(* 1 - During reseting, 0 - Reset completed
	Description:
		Reset the batetery replacement timer request.
		Indirectly resets the battery error. *) 
METHOD MR_BatteryReset : BOOL
IF NOT BatteryResetCompleted THEN
	bBusy 	:= TRUE;
	MR_BatteryReset := TRUE;
	BatteryReset :=	TRUE;
	fbMachineLogger.MR_AddLogs(CONCAT(sName,' : battery reset requested'));
	
ELSE 
	MR_BatteryReset := FALSE;
	BatteryReset :=	FALSE;
	bBusy 	:= FALSE;
	fbMachineLogger.MR_AddLogs(CONCAT(sName,' : battery reset done'));
	
END_IF
END_METHOD

(* 1 - Cycle paused, 0 - Cycle not paused
	Description:
		This method stop the program without reseting.
		IE. stops movement implicily 
		To restore the movement use MR_RestoreCycle or MR_GoHome *)
METHOD MR_CyclePause : BOOL
IF eCR800State = CR800_DOING_ACTION THEN
	bBusy 	:= TRUE;
	bCyclePause := TRUE;
	MR_CyclePause := FALSE;
	eCR800State := E_CR800State.CR800_CYCLE_PAUSING;
	fbMachineLogger.MR_AddLogs(CONCAT(sName,' : cycle pausing requested'));
	
ELSIF eCR800State = E_CR800State.CR800_CYCLE_PAUSING_DONE THEN
	bCyclePause	:= FALSE;
	MR_CyclePause := TRUE;
	bBusy 	:= FALSE;
	fbMachineLogger.MR_AddLogs(CONCAT(sName,' : cycle pausing done'));
	
END_IF
END_METHOD

(* 1 - During stopping, 0 - Cycle stop completed
	Description:
		This method stop the program, when the "End" command is met in the robots program.
		Caution: It stops the program AND reset it. To restore it you need to use MR_RestoreAuto. *) 

METHOD MR_CycleStop : BOOL
IF eCR800State = CR800_DOING_ACTION OR eCR800State = CR800_IDLE_CYCLE_PAUSED OR eCR800State = CR800_IDLE_AUTO_PAUSED THEN
	bBusy 	:= TRUE;
	bCycleStop 	:= TRUE;
	MR_CycleStop := FALSE;
	eCR800State := CR800_CYCLE_STOPPING;
	fbMachineLogger.MR_AddLogs(CONCAT(sName,' : cycle stopping requested'));
	
ELSIF eCR800State = CR800_CYCLE_STOPING_DONE THEN
	bDoAction := FALSE;
	bCycleStop := FALSE;
	MR_CycleStop := TRUE;
	bBusy 	:= FALSE;
	fbMachineLogger.MR_AddLogs(CONCAT(sName,' : cycle stopping done'));
	
END_IF
END_METHOD

(* 0 - Action not completed, 1 - Action completed
Description:
This method send request to do an action.
Robot will perform an action number that is called in input.
If the action is single and has and end use:
	IF MR_DoAction( iActionNumber := iExampleNumber) THEN
		bDO_A_FLIP := true ;
	END_IF
If the action is endless then just call it, and then use MR_CycleStop.
	MR_DoAction( iActionNumber := iExampleNumber) *)
METHOD MR_DoAction : BOOL
VAR_INPUT
	iActionNumber : UINT ;
END_VAR
IF eCR800State = CR800_IDLE_AUTO THEN
	IF iActionNumber <= 12 THEN 
		bError := TRUE ;
		eErrorID := CR800_ERROR_CANT_DO_SYSTEM_ACTION_IN_THIS_REQUEST ;
	ELSE
		bBusy 	:= TRUE;
		bDoAction := TRUE;
		bStopped := FALSE;
		MR_DoAction := FALSE;
		iActionNumber := iActionNumber;
		eCR800State := CR800_DOING_ACTION;
		fbMachineLogger.MR_AddLogs(FUN_MergeStrings5(sName,' : doing action number: ',UINT_TO_STRING(iActionNumber), '',' requested'));
	
	END_IF
	
ELSIF eCR800State = CR800_DOING_ACTION_DONE THEN
	bIsHomed := FALSE;
	bAutoModeStarted := FALSE;
	MR_DoAction := TRUE;
	bBusy := FALSE; 
	fbMachineLogger.MR_AddLogs(FUN_MergeStrings5(sName,' : doing action number: ',UINT_TO_STRING(iActionNumber),'',' done'));
	
ELSIF eCR800State <> CR800_DOING_ACTION AND eCR800State = E_CR800State.CR800_IDLE_CYCLE_PAUSED 
	AND eCR800State <> E_CR800State.CR800_CYCLE_PAUSING AND eCR800State <> E_CR800State.CR800_CYCLE_PAUSING
	AND eCR800State <> CR800_CYCLE_RESTORING AND eCR800State <> CR800_CYCLE_RESTORING_DONE THEN
	bError := TRUE ;
	eErrorID := CR800_ERROR_CANT_DO_ACTION_WITHOUT_BEEING_AUTO ;
	fbMachineLogger.MR_AddLogs(CONCAT(sName,' : ERROR_CANT_DO_ACTION_WITHOUT_BEEING_AUTO'));
	
END_IF
END_METHOD

METHOD MR_FirstCycle : BOOL
VAR_INPUT
	sName 				: STRING;
	iOverride			: USINT;
END_VAR
THIS^.sName := sName;
THIS^.iOverride := iOverride;
END_METHOD

(* 0 - FB is NOT in auto mode, 1 - FB is in auto mode
	Description:
		This method reqest FB to go into the auto mode. In automode FB can perform actions (MR_DoAction) *)
METHOD MR_GoAuto : BOOL
IF NOT bIsHomed THEN 
	bError := TRUE ;
	eErrorID := CR800_ERROR_CANT_GO_AUTO_WITHOUT_BEEING_HOMED ;
	fbMachineLogger.MR_AddLogs(CONCAT(sName,' : ERROR_CANT_GO_AUTO_WITHOUT_BEEING_HOMED'));
	
ELSIF eCR800State = CR800_IDLE_HOMED OR eCR800State = CR800_CYCLE_PAUSING_IDLE THEN
	bBusy 	:= TRUE;
	bGoAuto := TRUE;
	MR_GoAuto := FALSE;
	iActionNumber := stRobot.iActionNumber;
	eCR800State := CR800_GOING_AUTO;
	fbMachineLogger.MR_AddLogs(CONCAT(sName,' : going auto requested'));
	
ELSIF eCR800State = CR800_GOING_AUTO_DONE THEN
	bStopped := FALSE;
	bGoAuto := FALSE;
	MR_GoAuto := TRUE;
	bAutoModeStarted := TRUE;
	bBusy 	:= FALSE;
	fbMachineLogger.MR_AddLogs(CONCAT(sName,' : going auto done'));
	
END_IF
END_METHOD

(* 1 - Homing finished, 0 - Homing not finished.
	Description:
	This method request the robot to go home *)
METHOD MR_GoHome : BOOL
IF eCR800State = CR800_IDLE_NOT_HOMED OR eCR800State = CR800_IDLE_AUTO OR eCR800State = CR800_IDLE_AUTO_PAUSED THEN
	bBusy 	:= TRUE;	
	bGoHome := TRUE;
	MR_GoHome := FALSE;
	eCR800State := CR800_GOING_HOME;
	fbMachineLogger.MR_AddLogs(CONCAT(sName,' : going home requested'));
	
ELSIF eCR800State = CR800_GOING_HOME_DONE THEN
	bIsHomed := TRUE;
	bGoHome := FALSE;
	MR_GoHome := TRUE;
	bBusy 	:= FALSE;
	fbMachineLogger.MR_AddLogs(CONCAT(sName,' : going home done'));
	
END_IF
END_METHOD

(* 1 - Initializing finished, 0 - Initializing not finished.
	Description:
		This method initialize the robot:
			1. Checks for ethercat connection
			2. Checks for power of the CR800
			3. Checks for emergency stop
			4. Checks is CR800 is in auto mode
			5. Enable rights
			6. Turn on servos
			7. Resets the program
			8. Starts the program
			9. Sets initial parameters in the robot (when initializing after error this step is ommited) *)
METHOD MR_Init : BOOL
IF eCR800State = CR800_UNINITIALIZED AND NOT bAbort AND NOT bReset THEN
	bBusy 	:= TRUE;
	bInit := TRUE;
	MR_Init := FALSE;
	eCR800State := CR800_INITIALIZING;
	fbMachineLogger.MR_AddLogs(CONCAT(sName,' : initialization requested'));
	
ELSIF eCR800State = CR800_READY_INITIALIZED THEN
	bUninitialized := FALSE;
	bActive := TRUE;
	bInit := FALSE;
	MR_Init := TRUE;
	bBusy 	:= FALSE;
	fbMachineLogger.MR_AddLogs(CONCAT(sName,' : initialization done'));
	
END_IF
END_METHOD

(* 1 - Reset finished, 0 - Reset not finished.
	Description:
		This method resets the error state of the FB *)
METHOD MR_Reset : BOOL
IF eCR800State < CR800_RESET AND bError THEN
	bBusy 	:= TRUE;
	bReset := TRUE;
	eCR800StateBeforeReset := eCR800State;
	MR_Reset := FALSE;
	eCR800State := CR800_RESET;
	fbMachineLogger.MR_AddLogs(CONCAT(sName,' : reset requested'));
	
ELSIF eCR800State = CR800_RESET_DONE THEN
	bReset := FALSE;
	MR_Reset := TRUE;
	bBusy 	:= FALSE;
	fbMachineLogger.MR_AddLogs(CONCAT(sName,' : reset done'));
		
END_IF
END_METHOD

(* 1 - Reset finished, 0 - Reset not finished.
	Description:
		This method resets the internal error of CR800 *)
METHOD MR_ResetCR800Err : BOOL
IF ErrorOccuring  THEN
	bBusy 	:= TRUE;
	MR_ResetCR800Err := FALSE;
	ErrorReset := TRUE;
	fbMachineLogger.MR_AddLogs(CONCAT(sName,' : controller reset requested'));
	
ELSE 
	ErrorReset := FALSE;
	MR_ResetCR800Err := TRUE;	
	bBusy 	:= FALSE;
	fbMachineLogger.MR_AddLogs(CONCAT(sName,' : controller reset done'));
	
END_IF
END_METHOD

(* 1 - Auto mode restored, 0 - Auto mode NOT restored.
	Description:
		This method restores auto mode after the MR_CycleStop method *)
METHOD MR_RestoreAuto : BOOL
IF eCR800State = CR800_IDLE_AUTO_PAUSED THEN
	bBusy 	:= TRUE;
	bRestoreAuto := TRUE;
	bInitProgram := TRUE;
	MR_RestoreAuto := FALSE;
	eCR800State := CR800_AUTO_RESTORING;
	fbMachineLogger.MR_AddLogs(CONCAT(sName,' : restoring auto mode requested'));
	
ELSIF eCR800State = CR800_AUTO_RESTORING_DONE THEN
	bStopped := FALSE;
	bRestoreAuto := FALSE;
	bInitProgram := FALSE;
	MR_RestoreAuto := TRUE;
	bBusy 	:= FALSE;
	fbMachineLogger.MR_AddLogs(CONCAT(sName,' : restoring auto mode done'));
	
END_IF
END_METHOD

(* 1 - Cycle restored, 0 - Cycle NOT restored.
	Description:
		This method restores cycle after the MR_CyclePause method *)
METHOD MR_RestoreCycle : BOOL

VAR
	FA: BOOL;
END_VAR
IF eCR800State = CR800_IDLE_CYCLE_PAUSED THEN
	bBusy 	:= TRUE;
	bRestoreCycle := TRUE;
	MR_RestoreCycle	:= FALSE;
	eCR800State := CR800_CYCLE_RESTORING;
	fbMachineLogger.MR_AddLogs(CONCAT(sName,' : restoring cycle requested'));
		
ELSIF eCR800State = CR800_CYCLE_RESTORING_DONE THEN	
	bRestoreCycle := FALSE;
	MR_RestoreCycle := TRUE;
	bBusy 	:= FALSE;
	fbMachineLogger.MR_AddLogs(CONCAT(sName,' : restoring cycle done'));
	
END_IF
END_METHOD

METHOD MR_SendPosition1 : BOOL 
VAR_INPUT
	lrPositionX1	: LREAL;
	lrPositionY1	: LREAL;
	lrRotation1		: LREAL;
END_VAR
IF eCR800State = CR800_DOING_ACTION OR eCR800State = CR800_IDLE_AUTO_PAUSED OR eCR800State = CR800_IDLE_AUTO OR eCR800State = CR800_IDLE_HOMED OR eCR800State = CR800_IDLE_NOT_HOMED THEN
	bBusy 	:= TRUE;
	bSendPosition1 := TRUE;
	MR_SendPosition1 := FALSE;
	eCR800StateBeforeSendPosition := eCR800State;
	eCR800State := CR800_SEND_POSITION_1;
	eCR800StateSendPosition := CR800_SEND_POSITION_CONVERTING;
	THIS^.lrPositionX1 := lrPositionX1;
	THIS^.lrPositionY1 := lrPositionY1;
	THIS^.lrRotation1 := lrRotation1;
	fbMachineLogger.MR_AddLogs(CONCAT(sName,' : sending first position requested'));
	
ELSIF eCR800State = CR800_SEND_POSITION_1_DONE THEN
	bSendPosition1	:= FALSE;
	MR_SendPosition1 := TRUE;
	//bBusy := FALSE;
	fbMachineLogger.MR_AddLogs(CONCAT(sName,' : sending first position done'));
	
END_IF
END_METHOD

METHOD MR_SendPosition2 : BOOL 
VAR_INPUT
	lrPositionX2	: LREAL;
	lrPositionY2	: LREAL;
	lrRotation2		: LREAL;
END_VAR
IF eCR800State = CR800_DOING_ACTION OR eCR800State = CR800_IDLE_AUTO_PAUSED OR eCR800State = CR800_IDLE_AUTO OR eCR800State = CR800_IDLE_HOMED OR eCR800State = CR800_IDLE_NOT_HOMED THEN
	bBusy 	:= TRUE;
	bSendPosition2 := TRUE;
	MR_SendPosition2 := FALSE;
	eCR800StateBeforeSendPosition := eCR800State;
	eCR800State := CR800_SEND_POSITION_2;
	eCR800StateSendPosition := CR800_SEND_POSITION_CONVERTING;
	THIS^.lrPositionX2 := lrPositionX2;
	THIS^.lrPositionY2 := lrPositionY2;
	THIS^.lrRotation2 := lrRotation2;
	fbMachineLogger.MR_AddLogs(CONCAT(sName,' : sending second position requested'));
	
ELSIF eCR800State = CR800_SEND_POSITION_2_DONE THEN
	bSendPosition2	:= FALSE;
	MR_SendPosition2 := TRUE;
	//bBusy := FALSE;
	fbMachineLogger.MR_AddLogs(CONCAT(sName,' : sending second position done'));
	
END_IF
END_METHOD

(* 1 - Recipies updated, 0 - Recipies not updated.
	Description:
		This method updated the recipies, while robot is homed *)
METHOD MR_UpdateRecipies : BOOL
IF eCR800State = CR800_IDLE_HOMED THEN
	bBusy 	:= TRUE;
	bUpdateRecipes := TRUE;
	MR_UpdateRecipies := FALSE;
	eCR800State := CR800_UPDATING_RECIPIES;
	fbMachineLogger.MR_AddLogs(CONCAT(sName,' : updating recipes requested'));
	
ELSIF eCR800State = CR800_UPDATE_RECIPIES_DONE THEN
	bUpdateRecipes := FALSE;
	MR_UpdateRecipies := TRUE;
	bBusy 	:= FALSE;
	fbMachineLogger.MR_AddLogs(CONCAT(sName,' : updating recipes done'));
	
END_IF
END_METHOD

METHOD PROTECTED  MS_Aborting
CASE eCR800StateAbort OF
	
	CR800_ABORTING_IDLE:
		eCR800StateAbort := CR800_ABORTING_ENABLE_RIGHTS;
	
	CR800_ABORTING_ENABLE_RIGHTS:
		IF M_OperationRigtsEnable(bRequest := TRUE) THEN
			eCR800StateAbort := CR800_ABORTING_PRGM_STOP;
		END_IF
	
	CR800_ABORTING_PRGM_STOP: 
		IF M_ProgramStop() THEN
			eCR800StateAbort := CR800_ABORTING_PRGM_RESET ;
		END_IF
	
	CR800_ABORTING_PRGM_RESET: 
		IF M_ProgramReset() THEN
			IF NOT bInitProgram THEN
				eCR800StateAbort := CR800_ABORTING_SERVO_OFF ;
			ELSE 
				eCR800StateAbort := CR800_ABORTING_DONE ;
			END_IF
		END_IF
		
	CR800_ABORTING_SERVO_OFF: 
		IF M_ServoOFF() THEN
			eCR800StateAbort := CR800_ABORTING_DONE ;
		END_IF
	 
	CR800_ABORTING_DONE:
	
		M_OperationRigtsEnable(bRequest 	:= 0);
		eCR800StateDoRequest				:= 0 ;
		eCR800StateHome 					:= 0 ;	
		eCR800StateReceiveCommand			:= 0 ;
		eCR800SendCommand					:= 0 ;
		eCR800StateInitializing 			:= 0 ;
		eCR800StateCycleStop 				:= 0 ; 
		eCR800StateCyclePause				:= 0 ; 
		bGoHome 			:=	FALSE;
		bUpdateRecipes		:=	FALSE;
		bGoAuto				:=	FALSE;
		bDoAction			:=	FALSE;
		bCycleStop			:=	FALSE;
		bCyclePause			:= 	FALSE;
		bRestoreCycle		:=  FALSE;
		bIsHomed			:=	FALSE;
		bAutoModeStarted 	:=  FALSE;
		tonWatchdog.IN 		:=  FALSE;
		bInit				:= 	FALSE;
		
		IF NOT bInitProgram THEN
			eCR800State := CR800_UNINITIALIZED;
		ELSE 
			eCR800State := CR800_INITIALIZING;
		END_IF	
			
		eCR800StateAbort := CR800_ABORTING_IDLE ;
END_CASE
END_METHOD

METHOD PROTECTED MS_CyclePauseDone
IF NOT bCyclePause THEN
	eCR800State := CR800_IDLE_CYCLE_PAUSED ;
END_IF
END_METHOD

METHOD PROTECTED MS_CyclePausing
CASE eCR800StateCyclePause OF
	CR800_CYCLE_PAUSING_IDLE:
		eCR800StateCyclePause := E_CR800StateCyclePausing.CR800_CYCLE_PAUSING;
		
	E_CR800StateCyclePausing.CR800_CYCLE_PAUSING:
		IF M_ProgramStop() THEN
			eCR800StateCyclePause := E_CR800StateCyclePausing.CR800_CYCLE_PAUSING_DONE;
		END_IF
		
	E_CR800StateCyclePausing.CR800_CYCLE_PAUSING_DONE:
		eCR800State := E_CR800State.CR800_CYCLE_PAUSING_DONE;
		eCR800StateCyclePause := CR800_CYCLE_PAUSING_IDLE;
END_CASE
END_METHOD

METHOD PROTECTED MS_CycleStopDone
IF NOT bCycleStop THEN
	eCR800State := CR800_IDLE_AUTO_PAUSED ;
END_IF
END_METHOD

METHOD PROTECTED MS_CycleStopping
VAR_INST
	tonWait : TON := (pt := T#1S) ;
END_VAR
CASE eCR800StateCycleStop OF
	CR800_CYCLE_STOPPPING_IDLE:
		eCR800StateCycleStop := CR800_CYCLE_STOPPPING_SEND_REQUEST;
		
	CR800_CYCLE_STOPPPING_SEND_REQUEST:
		CycleStop := TRUE ;
		eCR800StateCycleStop := CR800_CYCLE_STOPPPING_WAIT_FOR_STOP;

	CR800_CYCLE_STOPPPING_WAIT_FOR_STOP:
		tonWait.IN := TRUE ;
		IF NOT CycleStopping AND tonWait.Q THEN
			eCR800StateCycleStop := CR800_CYCLE_STOPPPING_RESET_VARIABLES;
		END_IF
		
	CR800_CYCLE_STOPPPING_RESET_VARIABLES:
		tonWait.IN := FALSE ;
		bDoAction := FALSE;
		eCR800StateReceiveCommand := 0;
		eCR800SendCommand := 0;
		eCR800StateDoRequest := 0; 	
		eCR800StateCycleStop := CR800_CYCLE_STOPPPING_DONE;
		
	CR800_CYCLE_STOPPPING_DONE:
		CycleStop := FALSE ;
		eCR800State := CR800_CYCLE_STOPING_DONE;
		eCR800StateCycleStop := CR800_CYCLE_STOPPPING_IDLE ;
END_CASE

tonWait();
END_METHOD

METHOD PROTECTED MS_DoAction_Done
bDoAction := FALSE;
eCR800State := CR800_IDLE_AUTO ;
END_METHOD

METHOD PROTECTED MS_DoingAction
IF M_DoRequest(iNumberOfRequest := iActionNumber) THEN
	eCR800State := CR800_DOING_ACTION_DONE ;
END_IF
END_METHOD

METHOD PROTECTED MS_GoAutoDone
IF NOT bGoAuto THEN
	eCR800State := CR800_IDLE_AUTO ;
END_IF
END_METHOD

METHOD PROTECTED MS_GoHomeDone
IF NOT bGoHome THEN
	eCR800State := CR800_IDLE_HOMED ;
END_IF
END_METHOD

METHOD PROTECTED MS_GoingAuto
IF M_DoRequest(E_RobotSystemActions.GO_AUTO) THEN
	eCR800State := CR800_GOING_AUTO_DONE ;
END_IF
END_METHOD

METHOD PROTECTED MS_GoingHome
CASE eCR800StateHome OF

	CR800_HOMING_IDLE:
		IF eCR800State = CR800_IDLE_AUTO OR eCR800State = CR800_IDLE_AUTO_PAUSED THEN
			eCR800StateHome	:= CR800_HOMING_RESET_PROGRAM ;
		ELSE 
			eCR800StateHome	:= CR800_HOMING_SEND_REQUEST ;
		END_IF
		
	CR800_HOMING_RESET_PROGRAM:
		IF M_ProgramReset() THEN
			eCR800StateHome := CR800_HOMING_RESET_CYCLE_VARIABLES ;
		END_IF	
		
	CR800_HOMING_RESET_CYCLE_VARIABLES:
		bDoAction := FALSE;
		eCR800StateReceiveCommand := 0;
		eCR800SendCommand := 0;
		eCR800StateDoRequest := 0;
		eCR800StateHome := CR800_HOMING_START_PROGRAM ;	
	
		
	CR800_HOMING_START_PROGRAM:
		IF M_ProgramStart() THEN
			eCR800StateHome := CR800_HOMING_SEND_REQUEST ;
		END_IF
	
	CR800_HOMING_SEND_REQUEST:
		IF M_DoRequest(E_RobotSystemActions.DO_HOMING) THEN   
			eCR800StateHome := CR800_HOMING_DONE ;
		END_IF	
		
	CR800_HOMING_DONE:
		eCR800State := CR800_GOING_HOME_DONE ;
		eCR800StateHome := CR800_HOMING_IDLE ;
END_CASE
END_METHOD

METHOD PROTECTED MS_IdleAuto
;
END_METHOD

METHOD PROTECTED MS_IdleAutoPaused
;
END_METHOD

METHOD PROTECTED MS_IdleCyclePaused
;
END_METHOD

METHOD PROTECTED MS_IdleHomed
;
END_METHOD

METHOD PROTECTED MS_IdleNotHomed
;
END_METHOD

METHOD PROTECTED MS_InExternalError
bDontSetInitialParameters := TRUE;
END_METHOD

METHOD PROTECTED MS_Initializing
CASE eCR800StateInitializing OF
		
	CR800_INIT_IDLE:
		eCR800StateInitializing := CR800_INIT_ETHERCAT_CHCEK ;
		
	CR800_INIT_ETHERCAT_CHCEK:
		tonWatchdog.IN := TRUE ;
		IF stCR800EthercatData.iInfoDataState = 8 THEN
			tonWatchdog.IN := FALSE ;	
			eCR800StateInitializing := CR800_INIT_POWER_CHCECK;
		ELSIF tonWatchdog.Q THEN
			bError := TRUE ;
			eErrorID := CR800_ERROR_ETHERCAT_CHECK_FAIL ;			
		END_IF
	
	CR800_INIT_POWER_CHCECK:
		tonWatchdog.IN := TRUE ;
		IF CR800PoweredOn THEN
			tonWatchdog.IN := FALSE ;	
			eCR800StateInitializing := CR800_INIT_EMERG_STOP_CHCECK;
		ELSIF tonWatchdog.Q THEN
			bError := TRUE ;
			eErrorID := CR800_ERROR_POWER_CHECK_FAIL ;			
		END_IF
		
		
	CR800_INIT_EMERG_STOP_CHCECK:
		tonWatchdog.IN := TRUE ;
		IF NOT EmergencyStopOccuring THEN
			tonWatchdog.IN := FALSE ;	
			eCR800StateInitializing := CR800_INIT_CHECK_FOR_AUTO_MODE;
		ELSIF tonWatchdog.Q THEN
			bError := TRUE ;
			eErrorID := CR800_ERROR_EMERGENCY_STOP_OCCURING ;			
		END_IF
		
	CR800_INIT_CHECK_FOR_AUTO_MODE:
		tonWatchdog.IN := TRUE;
		IF InAutomaticMode THEN
			tonWatchdog.IN 			:= FALSE ;	
			eCR800StateInitializing := CR800_INIT_ENABLE_RIGHTS;
		ELSIF tonWatchdog.Q THEN
			bError := TRUE ;
			eErrorID := CR800_ERROR_AUTO_MODE_CHECK_FAIL ;		
		END_IF
		
	CR800_INIT_ENABLE_RIGHTS:
		IF M_OperationRigtsEnable(bRequest := TRUE) THEN
			eCR800StateInitializing	:= CR800_INIT_SERVO_ON ;
		END_IF
		
	CR800_INIT_SERVO_ON:
		IF M_ServoON() THEN
			eCR800StateInitializing	:= CR800_INIT_PROGRAM_RESET ;
		END_IF
		
	CR800_INIT_PROGRAM_RESET:
		IF M_ProgramReset() THEN
			eCR800StateInitializing	:= CR800_INIT_PROGRAM_START ;
		END_IF
			
	CR800_INIT_PROGRAM_START:
		IF M_ProgramStart() THEN
			IF bDontSetInitialParameters THEN 
				bDontSetInitialParameters := FALSE ;
				eCR800StateInitializing := CR800_INIT_DONE ;			
			ELSE
				eCR800StateInitializing := CR800_INIT_SET_INITIAL_PARAMETERS_REQUEST ;				
			END_IF
		END_IF	

	CR800_INIT_SET_INITIAL_PARAMETERS_REQUEST: 
		IF M_DoRequest(iNumberOfRequest := E_RobotSystemActions.SET_INITIAL_PARAMETERS) THEN
			eCR800StateInitializing := CR800_INIT_DONE ;
		END_IF

	CR800_INIT_DONE:
		IF NOT bInitProgram THEN
			eCR800State := CR800_READY_INITIALIZED;
		ELSE
			eCR800State := CR800_AUTO_RESTORING_DONE;
		END_IF
		eCR800StateInitializing := CR800_INIT_IDLE ;
			
END_CASE
END_METHOD

METHOD PROTECTED MS_ReadyInitialized
VAR_INPUT
END_VAR
eCR800State := CR800_IDLE_NOT_HOMED;
END_METHOD

METHOD PROTECTED MS_Reset
VAR_INPUT
END_VAR
M_ResetVariables();
IF MR_ResetCR800Err() THEN
	eCR800State := CR800_RESET_DONE;
	eErrorID := CR800_ERROR_OK;
	bError := FALSE;
END_IF
END_METHOD

METHOD PROTECTED MS_ResetDone
VAR_INPUT
END_VAR
IF NOT bReset THEN
	IF eCR800StateBeforeReset >= CR800_IDLE_NOT_HOMED  THEN
		eCR800State := CR800_IDLE_NOT_HOMED ;
	ELSE
		eCR800State := CR800_UNINITIALIZED ;
	END_IF
END_IF
END_METHOD

METHOD PROTECTED MS_RestoreAutoDone
IF NOT bRestoreAuto THEN
	eCR800State := CR800_IDLE_NOT_HOMED ;
END_IF
END_METHOD

METHOD PROTECTED MS_RestoreCycleDone
IF NOT bRestoreCycle THEN
	eCR800State := CR800_DOING_ACTION ;
END_IF
END_METHOD

METHOD PROTECTED MS_RestoringAuto
eCR800State := CR800_ABORTING ;
END_METHOD

METHOD PROTECTED MS_RestoringCycle
IF M_ProgramStart() THEN 
	eCR800State := CR800_CYCLE_RESTORING_DONE ;
END_IF
END_METHOD

METHOD PROTECTED MS_SendingPosition1
VAR_INST
	lrPositionXFirstHalf  	: LREAL;
	lrPositionXSecondHalf  	: LREAL;
	lrPositionYFirstHalf  	: LREAL;
	lrPositionYSecondHalf 	: LREAL;
	lrRotationFirstHalf  	: LREAL;
	lrRotationSecondHalf	: LREAL;
END_VAR
CASE eCR800StateSendPosition OF 
	CR800_SEND_POSITION_CONVERTING:
		LTRUNC( lr_in := lrPositionX1,
				LTRUNC => lrPositionXFirstHalf);
		LTRUNC( lr_in := lrPositionY1,
				LTRUNC => lrPositionYFirstHalf);
		LTRUNC( lr_in := lrRotation1,
				LTRUNC => lrRotationFirstHalf);
	
		FRAC( lr_in := lrPositionX1,
				FRAC => lrPositionXSecondHalf);
		FRAC( lr_in := lrPositionY1,
				FRAC => lrPositionYSecondHalf);
		FRAC( lr_in := lrRotation1,
				FRAC => lrRotationSecondHalf);
				
		eCR800StateSendPosition := CR800_SEND_POSITION_SENDING;
		
	CR800_SEND_POSITION_SENDING:
		stCR800EthercatData.arrRegistersOutput[6022] :=	LREAL_TO_INT(lrPositionXFirstHalf); 
		stCR800EthercatData.arrRegistersOutput[6023] :=	LREAL_TO_INT(1000 * lrPositionXSecondHalf); 
		stCR800EthercatData.arrRegistersOutput[6024] :=	LREAL_TO_INT(lrPositionYFirstHalf); 
		stCR800EthercatData.arrRegistersOutput[6025] :=	LREAL_TO_INT(1000 * lrPositionYSecondHalf); 
		stCR800EthercatData.arrRegistersOutput[6026] :=	LREAL_TO_INT(lrRotationFirstHalf); 
		stCR800EthercatData.arrRegistersOutput[6027] :=	LREAL_TO_INT(1000 * lrRotationSecondHalf); 
			
		eCR800State := CR800_SEND_POSITION_1_DONE;
		
END_CASE
END_METHOD

METHOD PROTECTED MS_SendingPosition1Done
IF NOT bSendPosition1 THEN
	eCR800State := eCR800StateBeforeSendPosition;
	bBusy := FALSE;
	
END_IF
END_METHOD

METHOD PROTECTED MS_SendingPosition2
VAR_INST
	lrPositionXFirstHalf  	: LREAL;
	lrPositionXSecondHalf  	: LREAL;
	lrPositionYFirstHalf  	: LREAL;
	lrPositionYSecondHalf 	: LREAL;
	lrRotationFirstHalf  	: LREAL;
	lrRotationSecondHalf	: LREAL;
END_VAR
CASE eCR800StateSendPosition OF 
	CR800_SEND_POSITION_CONVERTING:
		LTRUNC( lr_in := lrPositionX2,
				LTRUNC => lrPositionXFirstHalf);
		LTRUNC( lr_in := lrPositionY2,
				LTRUNC => lrPositionYFirstHalf);
		LTRUNC( lr_in := lrRotation2,
				LTRUNC => lrRotationFirstHalf);
	
		FRAC( lr_in := lrPositionX2,
				FRAC => lrPositionXSecondHalf);
		FRAC( lr_in := lrPositionY2,
				FRAC => lrPositionYSecondHalf);
		FRAC( lr_in := lrRotation2,
				FRAC => lrRotationSecondHalf);
				
		eCR800StateSendPosition := CR800_SEND_POSITION_SENDING;
		
	CR800_SEND_POSITION_SENDING:
		stCR800EthercatData.arrRegistersOutput[6028] :=	LREAL_TO_INT(lrPositionXFirstHalf); 
		stCR800EthercatData.arrRegistersOutput[6029] :=	LREAL_TO_INT(1000 * lrPositionXSecondHalf); 
		stCR800EthercatData.arrRegistersOutput[6030] :=	LREAL_TO_INT(lrPositionYFirstHalf); 
		stCR800EthercatData.arrRegistersOutput[6031] :=	LREAL_TO_INT(1000 * lrPositionYSecondHalf); 
		stCR800EthercatData.arrRegistersOutput[6032] :=	LREAL_TO_INT(lrRotationFirstHalf); 
		stCR800EthercatData.arrRegistersOutput[6033] :=	LREAL_TO_INT(1000 * lrRotationSecondHalf); 
			
		eCR800State := CR800_SEND_POSITION_2_DONE;
		
END_CASE
END_METHOD

METHOD PROTECTED MS_SendingPosition2Done
IF NOT bSendPosition2 THEN
	eCR800State := eCR800StateBeforeSendPosition;
	bBusy := FALSE;
	
END_IF
END_METHOD

METHOD Protected MS_Uninitialized
VAR_inst
	iLoop: INT;
END_VAR
//M_ResetVariables();

//M_OperationRigtsEnable(bRequest 	:= 0);
//eCR800StateDoRequest				:= 0 ;
eCR800StateHome 					:= 0 ;	
//eCR800StateReceiveCommand			:= 0 ;
//eCR800SendCommand					:= 0 ;
//eCR800StateInitializing 			:= 0 ;
eCR800StateCycleStop 				:= 0 ; 
eCR800StateCyclePause				:= 0 ; 
eCR800StateSendPosition				:= 0 ;

eErrorID := CR800_ERROR_OK;

bUninitialized := TRUE;
bInit := FALSE;
bGoHome := FALSE;
bUpdateRecipes := FALSE;
bGoAuto := FALSE;
bDoAction := FALSE;
bCycleStop := FALSE;
bCyclePause := FALSE;
bRestoreAuto := FALSE;
bRestoreCycle := FALSE;
bAbort := FALSE;
bError := FALSE;
bAutoModeStarted := FALSE;
bIsHomed := FALSE;
bReset := FALSE;
bStopped := FALSE;
bActive := FALSE; 
	
IF ServoIsOn THEN
	MR_Abort();
END_IF
END_METHOD

METHOD PROTECTED MS_UpdateRecipiesDone
IF NOT bUpdateRecipes THEN
	eCR800State := CR800_IDLE_HOMED ;
END_IF
END_METHOD

METHOD PROTECTED MS_UpdatingRecipies
IF M_DoRequest(iNumberOfRequest := E_RobotSystemActions.UPDATE_RECIPIES) THEN
	eCR800State := CR800_UPDATE_RECIPIES_DONE ;
END_IF
END_METHOD

PROPERTY Name : STRING
GET
Name := sName;
END_GET
SET
sName := Name;
END_SET
END_PROPERTY

(* Desription from CR800 side: Sets the validity of the operation rights for the
external signal control.. *)
{attribute 'monitoring' := 'variable'}
PROPERTY OperationRightsEnable : BOOL
GET
OperationRightsEnable := stCR800EthercatData.arrSignalsOutputConverted[6004] ;
END_GET
SET
stCR800EthercatData.arrSignalsOutputConverted[6004] := OperationRightsEnable ;
END_SET
END_PROPERTY

(*Desription from CR800 side:
Outputs the operation rights valid state for the
external signal control.
The operation right is given when the
operation right input signal is ON, the
controller mode is set to AUTOMATIC, and
there is no other device that currently has the
operation right.*)
{attribute 'monitoring' := 'variable'}
PROPERTY PUBLIC OperationRightsEnabled : BOOL
GET
OperationRightsEnabled := stCR800EthercatData.arrSignalsInputConverted[6004] ;
END_GET
END_PROPERTY

(* Reqest number that robot has to perform *)
{attribute 'monitoring' := 'variable'}
PROPERTY Override : USINT
GET
//Override :=	INT_TO_USINT(stCR800EthercatData.arrRegistersOutput[6021]);
Override := iOverride;
END_GET
SET
//stCR800EthercatData.arrRegistersOutput[6021] := USINT_TO_INT(iOverride);
iOverride := Override;
END_SET
END_PROPERTY

(* Desription from CR800 side:
"This output indicates that the program is
paused.
Turns ON when there is not slot multitask
running, and at least one slot is pausing.
However, slots whose starting condition is set
to ALWAYS or ERROR via a parameter
""SLT**"" will not be executed." *)
{attribute 'monitoring' := 'variable'}
PROPERTY PUBLIC Pausing : BOOL
GET
Pausing := stCR800EthercatData.arrSignalsInputConverted[6006] ;
END_GET
END_PROPERTY

(* Desription from CR800 side:
"This output indicates that a program is being
executed. During multitask operation, this
signal turns ON when at least one task slot is
operating.
However, slots whose starting condition is set
to ALWAYS or ERROR via a parameter ""SLT*""
will not be executed." *)
{attribute 'monitoring' := 'variable'}
PROPERTY PUBLIC ProgramOperating : BOOL
GET
ProgramOperating := stCR800EthercatData.arrSignalsInputConverted[6005] ;
END_GET
END_PROPERTY

(* Desription from CR800 side:
"This input cancels the paused status of the
program and brings the executing line to the
top. Executing a program reset makes it
possible to select a program.
In the multitask mode, the program reset is
applied to all task slots.
However, slots whose starting condition is set
to ALWAYS or ERROR via a parameter
""SLT**"" will not be executed." *)
{attribute 'monitoring' := 'variable'}
PROPERTY ProgramReset : BOOL
GET
ProgramReset := stCR800EthercatData.arrSignalsOutputConverted[6009] ;
END_GET
SET
stCR800EthercatData.arrSignalsOutputConverted[6009] := ProgramReset ;
END_SET
END_PROPERTY

(* "Outputs that in the program selection enabled
state.
Turns ON when program are not running or
pausing.
In multitask operation, this output turns ON
when all task slots are neither operating nor
paused.
However, slots whose starting condition is set
to ALWAYS or ERROR via a parameter
""SLT**"" will not be executed" *)
{attribute 'monitoring' := 'variable'}
PROPERTY PUBLIC ProgramSelectionEnabled : BOOL
GET
ProgramSelectionEnabled := stCR800EthercatData.arrSignalsInputConverted[6009] ;
END_GET
END_PROPERTY

(*Desription from CR800 side:
"This input starts a program. To start a specific
program, select the program using the
program selection signal ""PRGSEL"" and
numerical input ""IODATA,"" and then input the
start signal. Note that when the parameter
""PST"" is enabled, the system reads the
program number from the numerical input
(IODATA) and starts the corresponding
program (i.e., program selection becomes no
longer necessary).
All task slots are executed during multitask
operation.
However, slots whose starting condition is set
to ALWAYS or ERROR via a parameter ""SLT*""
will not be executed." *)
{attribute 'monitoring' := 'variable'}
PROPERTY ProgramStart : BOOL ;
GET
ProgramStart := stCR800EthercatData.arrSignalsOutputConverted[6005] ;
END_GET
SET
stCR800EthercatData.arrSignalsOutputConverted[6005] := ProgramStart ;
END_SET
END_PROPERTY

(* Desription from CR800 side:
This input stops the program being executed.
(The specification is the same as for the STOP
parameter.)
Unlike the STOP parameter, signal numbers
can be changed. *)
{attribute 'monitoring' := 'variable'}
PROPERTY ProgramStop2 : BOOL
GET
ProgramStop2 := stCR800EthercatData.arrSignalsOutputConverted[6007] ;
END_GET
SET
stCR800EthercatData.arrSignalsOutputConverted[6007] := ProgramStop2 ;
END_SET
END_PROPERTY

(* Desription from CR800 side:
"This output indicates that the program is
paused.
(The specification is the same as for the STOP
parameter.)" *)
{attribute 'monitoring' := 'variable'}
PROPERTY PUBLIC ProgramStopped : BOOL
GET
ProgramStopped := bStopped; // stCR800EthercatData.arrSignalsInputConverted[6007] ;
END_GET
END_PROPERTY

(* Reqest number that robot has to perform *)
{attribute 'monitoring' := 'variable'}
PROPERTY RequestNumber : UINT
GET
RequestNumber := iActionNumber;
END_GET
SET
stCR800EthercatData.arrRegistersOutput[6010] :=	UINT_TO_INT(RequestNumber);
END_SET
END_PROPERTY

PROPERTY SendingPosition1 : REFERENCE TO BOOL
GET
SendingPosition1 REF= bSendPosition1;
END_GET
END_PROPERTY

PROPERTY SendingPosition2 : REFERENCE TO BOOL
GET
SendingPosition2 REF= bSendPosition2;
END_GET
END_PROPERTY

(* Desription from a CR800 side:
"This input turns OFF the servo power supply
for the robot.(Applicable to all mechanisms)
The servo cannot be turned ON while this
signal is being input. *)
{attribute 'monitoring' := 'variable'}
PROPERTY PUBLIC ServoIsOff : BOOL
GET
ServoIsOff := NOT ServoIsOn AND CR800PoweredOn; //stCR800EthercatData.arrSignalsInputConverted[6012] ;
END_GET
END_PROPERTY

(* Desription from the CR800 side:
"This output turns ON when the servo power
supply for the robot is ON. If the servo power
supply is OFF, this output also remains OFF.
With a multi-mechanism configuration, this
output turns ON when the servo of at least one
mechanism is ON." *)
{attribute 'monitoring' := 'variable'}
PROPERTY PUBLIC ServoIsOn : BOOL
GET
ServoIsOn := stCR800EthercatData.arrSignalsInputConverted[6011] ;
END_GET
END_PROPERTY

(* Desription from a CR800 side:
"This input turns OFF the servo power supply
for the robot.(Applicable to all mechanisms)
The servo cannot be turned ON while this
signal is being input." *)
{attribute 'monitoring' := 'variable'}
PROPERTY ServoOFF : BOOL
GET
ServoOFF := stCR800EthercatData.arrSignalsOutputConverted[6012] ;
END_GET
SET
stCR800EthercatData.arrSignalsOutputConverted[6012] := ServoOFF ;
END_SET
END_PROPERTY

(* Descrition from the CR800 side:
"This input turns ON the servo power supply for
the robot.
With a multi-mechanism configuration, the
servo power supplies for all mechanisms will
be turned ON." *)
{attribute 'monitoring' := 'variable'}
PROPERTY ServoON : BOOL
GET
ServoON := stCR800EthercatData.arrSignalsOutputConverted[6011] ;
END_GET
SET
stCR800EthercatData.arrSignalsOutputConverted[6011] := ServoON ;
END_SET
END_PROPERTY

(* Actual state of main state machine *)
{attribute 'monitoring' := 'variable'}
PROPERTY State : REFERENCE TO E_CR800State
GET
State REF= eCR800State;
END_GET
END_PROPERTY

METHOD Protected StateMachine
VAR
	MS_CycleStopping_Done: INT;
END_VAR
CASE eCR800State OF
	CR800_UNINITIALIZED:
		MS_Uninitialized();
		
	CR800_INITIALIZING:
		MS_Initializing();
		
	CR800_READY_INITIALIZED:
		MS_ReadyInitialized();

	CR800_IDLE_NOT_HOMED:
		MS_IdleNotHomed();
		
	CR800_GOING_HOME:
		MS_GoingHome();
	
	CR800_GOING_HOME_DONE:
		MS_GoHomeDone();
		
	CR800_IDLE_HOMED:
		MS_IdleHomed();

	CR800_UPDATING_RECIPIES	:
		MS_UpdatingRecipies();
		
	CR800_UPDATE_RECIPIES_DONE:
		MS_UpdateRecipiesDone();
		
	CR800_GOING_AUTO:
		MS_GoingAuto();
		
	CR800_GOING_AUTO_DONE:
		MS_GoAutoDone();
		
	CR800_IDLE_AUTO:
		MS_IdleAuto();
		
	CR800_DOING_ACTION:
		MS_DoingAction();
		
	CR800_DOING_ACTION_DONE:
		MS_DoAction_Done();

	CR800_CYCLE_STOPPING:	
		MS_CycleStopping();
		
	CR800_CYCLE_STOPING_DONE:
		MS_CycleStopDone();
		
	CR800_IDLE_AUTO_PAUSED:
		MS_IdleAutoPaused();
		
	CR800_AUTO_RESTORING:
		MS_RestoringAuto();
	
	CR800_AUTO_RESTORING_DONE:
		MS_RestoreAutoDone();
		
	E_CR800State.CR800_CYCLE_PAUSING:
		MS_CyclePausing();
		
	E_CR800State.CR800_CYCLE_PAUSING_DONE:
		MS_CyclePauseDone();
	
	CR800_IDLE_CYCLE_PAUSED:
		MS_IdleCyclePaused();
	
	CR800_CYCLE_RESTORING:
		MS_RestoringCycle();
	
	CR800_CYCLE_RESTORING_DONE:
		MS_RestoreCycleDone();

	CR800_IN_EXTERNAL_ERROR:
		MS_InExternalError();
		
	CR800_SEND_POSITION_1:
		MS_SendingPosition1();
	
	CR800_SEND_POSITION_1_DONE:
		MS_SendingPosition1Done();	
		
	CR800_SEND_POSITION_2:
		MS_SendingPosition2();
	
	CR800_SEND_POSITION_2_DONE:
		MS_SendingPosition2Done();			
		
	CR800_RESET:
		MS_Reset();
		
	CR800_RESET_DONE:
		MS_ResetDone();
		
	CR800_ABORTING:
		MS_Aborting();
					
END_CASE
END_METHOD

(* Desription from CR800 side:
"Outputs that the stop is being input. (Logical
ADD of all devices.)" *)
{attribute 'monitoring' := 'variable'}
PROPERTY PUBLIC StopSTS : BOOL
GET
StopSTS := stCR800EthercatData.arrSignalsInputConverted[6008] ;
END_GET
END_PROPERTY

PROPERTY Uninitialized : REFERENCE TO BOOL
GET
Uninitialized REF= bUninitialized;
END_GET
END_PROPERTY

(*Desription from CR800 side:
This output indicates that the controller mode
is set to AUTOMATIC.*)
{attribute 'monitoring' := 'variable'}
{attribute 'monitoring' := 'call'}
PROPERTY  UserDefinedArea : ST_CR800UserDefinedArea
GET
UserDefinedArea.bArea1 := stCR800EthercatData.arrSignalsInputConverted[6241];
UserDefinedArea.bArea2 := stCR800EthercatData.arrSignalsInputConverted[6242];
UserDefinedArea.bArea3 := stCR800EthercatData.arrSignalsInputConverted[6243];
UserDefinedArea.bArea4 := stCR800EthercatData.arrSignalsInputConverted[6244];
UserDefinedArea.bArea5 := stCR800EthercatData.arrSignalsInputConverted[6245];
UserDefinedArea.bArea6 := stCR800EthercatData.arrSignalsInputConverted[6246];
UserDefinedArea.bArea7 := stCR800EthercatData.arrSignalsInputConverted[6247];
UserDefinedArea.bArea8 := stCR800EthercatData.arrSignalsInputConverted[6248];
END_GET
END_PROPERTY

PROPERTY UserDefinedArea1 : BOOL
GET
UserDefinedArea1 := stCR800EthercatData.arrSignalsInputConverted[6241];
END_GET
END_PROPERTY

PROPERTY UserDefinedArea2 : BOOL
GET
UserDefinedArea2 := stCR800EthercatData.arrSignalsInputConverted[6242];
END_GET
END_PROPERTY

PROPERTY UserDefinedArea3 : BOOL
GET
UserDefinedArea3 := stCR800EthercatData.arrSignalsInputConverted[6243];
END_GET
END_PROPERTY

PROPERTY UserDefinedArea4 : BOOL
GET
UserDefinedArea4 := stCR800EthercatData.arrSignalsInputConverted[6244];
END_GET
END_PROPERTY

PROPERTY UserDefinedArea5 : BOOL
GET
UserDefinedArea5 := stCR800EthercatData.arrSignalsInputConverted[6245];
END_GET
END_PROPERTY

PROPERTY UserDefinedArea6 : BOOL
GET
UserDefinedArea6 := stCR800EthercatData.arrSignalsInputConverted[6246];
END_GET
END_PROPERTY

PROPERTY UserDefinedArea7 : BOOL
GET
UserDefinedArea7 := stCR800EthercatData.arrSignalsInputConverted[6247];
END_GET
END_PROPERTY

PROPERTY UserDefinedArea8 : BOOL
GET
UserDefinedArea8 := stCR800EthercatData.arrSignalsInputConverted[6248];
END_GET
END_PROPERTY

END_FUNCTION_BLOCK

// ---- POUs/Libs/Utilities/File Logger/FB_FileLogger.TcPOU
(* 
:Description: This function block allows to log the data to txt file
*)
FUNCTION_BLOCK FB_FileLogger IMPLEMENTS I_FileLogger
VAR CONSTANT
	iBUFFER_SIZE : UINT := 255;
END_VAR
VAR
	sName : STRING;
	
	(* First cycle bits used for selecting file logging mode *)
	bAddTimeStamp				: BOOL;
	bAddHeader					: BOOL;
	
	(* Internal status *)
	bActive 					: BOOL;						(*  *)
	bBusy						: BOOL;						(*  *)
	bError						: BOOL;						(*  *)
	iErrorID					: UDINT;					(*  *)
	
	eFileLoggerState 			: E_FileLoggerState;		(*  *)
	eFileLoggerInitState 		: E_FileLoggerInitState;	(*  *)
	eFileLoggerAddLogsState		: E_FileLoggerAddLogsState; (*  *)
	eFileLoggerSetNewPathState 	: E_FileLoggerSetNewPathState;
	
	(* Internal parameters *)
	sFileName 					: STRING;					(*  *)
	sFileDir					: STRING;					(*  *)
	sFilePath					: STRING;					(*  *)
	
	hFile						: UINT;						(*  *)
	sAmsNetId					: T_AmsNetID;				(*  *)
	stTime						: TIMESTRUCT;				(*  *)
	sTime						: STRING;					(*  *)
	sFileDate					: STRING;									(*  *)
	sLogMessage					: STRING;									(*  *)
	
	(* Buffer arrays *)
	iCurrentBufferLine			: UINT := 1;								(*  *)
	iCurrentBufferLineForFile	: UINT := 1;								(*  *)
	arrMessageBuffer 			: ARRAY [1..iBUFFER_SIZE] OF STRING(300);	(*  *)
	arrMessageBufferPresence	: ARRAY [1..iBUFFER_SIZE] OF BOOL(255);		(*  *)
	
	(* Function blocks - time handling*)
	//fbGetTime					: NT_GetTime;				(*  *)
	
	(* Function blocks - file handling *)
	fbFileOpen					: FB_FileOpen;				(*  *)
	fbFileClose					: FB_FileClose;				(*  *)
	fbCreateDir					: FB_CreateDir;				(*  *)
	fbFilePuts					: FB_FilePuts;				(*  *)
END_VAR

bActive := eFileLoggerState >= FILE_LOGGER_READY;

IF fbMachineTime.bValid THEN
	stTime := fbMachineTime.systemTime;
	sTime := SYSTEMTIME_TO_STRING(stTime);
	
END_IF

StateMachine();

PROPERTY Active : REFERENCE TO BOOL
GET
Active REF= bActive;
END_GET
END_PROPERTY

PROPERTY AmsNetId : STRING
GET
AmsNetID := sAmsNetId;
END_GET
SET
sAmsNetId := AmsNetId;
END_SET
END_PROPERTY

PROPERTY Busy : REFERENCE TO BOOL
GET
Busy REF= bBusy;
END_GET
END_PROPERTY

PROPERTY Error : REFERENCE TO BOOL
GET
Error REF= bError;
END_GET
END_PROPERTY

PROPERTY ErrorID : REFERENCE TO UDINT
GET
ErrorID REF= iErrorID;
END_GET
END_PROPERTY

PROPERTY FileDir : STRING
GET
FileDir := sFileDir;
END_GET
SET
sFileDir := FileDir;
END_SET
END_PROPERTY

PROPERTY FileName : STRING
GET
FileName := sFileName;
END_GET
SET
sFileName := FileName;
END_SET
END_PROPERTY

METHOD M_ResetParameters : BOOL
VAR_INPUT
END_VAR
fbCreateDir( bExecute := FALSE);
fbFileOpen( bExecute := FALSE);
fbFilePuts( bExecute := FALSE);
fbFileClose( bExecute := FALSE);

FOR iCurrentBufferLine := 1 TO iBUFFER_SIZE BY 1 DO
	MEMSET(ADR(arrMessageBuffer[iCurrentBufferLine]),0,SIZEOF(arrMessageBuffer[iCurrentBufferLine]));
	arrMessageBufferPresence[iCurrentBufferLine] := FALSE;
END_FOR

iCurrentBufferLine := 1;
iCurrentBufferLineForFile := 1;

bError 		:= FALSE;
iErrorID 	:= 0;

MEMSET(ADR(sLogMessage),0,SIZEOF(sLogMessage));

eFileLoggerInitState := 0;
eFileLoggerAddLogsState := 0;
END_METHOD

METHOD M_SetNewPath : BOOL
VAR_INPUT
END_VAR
CASE eFileLoggerSetNewPathState OF
	FILE_LOGGER_SET_NEW_PATH_CHANGE_PATH:
		M_SetNewPath := FALSE;
		sFilePath := CONCAT(STR1 := sFileDir, STR2 := sFileName);
		
		eFileLoggerSetNewPathState := FILE_LOGGER_SET_NEW_PATH_DONE;
	
	FILE_LOGGER_SET_NEW_PATH_DONE:
		M_SetNewPath := TRUE;
		eFileLoggerSetNewPathState := FILE_LOGGER_SET_NEW_PATH_CHANGE_PATH;
			
END_CASE
END_METHOD

METHOD MR_Abort : BOOL
IF eFileLoggerState >= FILE_LOGGER_READY THEN
	bBusy := TRUE;
	MR_Abort := FALSE;
	eFileLoggerState := FILE_LOGGER_ABORTING;
	
ELSIF eFileLoggerState = FILE_LOGGER_UNINITIALIZED THEN
	bBusy := FALSE;
	MR_Abort := TRUE;
	
END_IF
END_METHOD

METHOD MR_AddLogs : BOOL
VAR_INPUT
	sLogMessage 	: STRING;		
	
END_VAR
VAR
	sCurrentTime 	: STRING;
	sCurrentDate	: STRING;
	sLog			: STRING(300);
	
END_VAR
IF iCurrentBufferLine >= iBUFFER_SIZE THEN	
	iCurrentBufferLine := 1;
		
ELSE
	sCurrentDate := LEFT(sTime,10);
	sCurrentTime := RIGHT(sTime,12);
	MEMSET(ADR(sLog),0,SIZEOF(sLog));
	
	IF bAddTimeStamp THEN
		sLog := FUN_MergeStrings6(sCurrentDate,'$t',sCurrentTime,'$t',sLogMessage,'$n'); 
	ELSE
		sLog := CONCAT(sLogMessage,'$n'); 
	END_IF
	
	MEMSET(ADR(arrMessageBuffer[iCurrentBufferLine]),0,SIZEOF(arrMessageBuffer[iCurrentBufferLine]));
	arrMessageBuffer[iCurrentBufferLine] := sLog;
	iCurrentBufferLine := iCurrentBufferLine + 1;
	
	MR_AddLogs := TRUE;
	
END_IF
END_METHOD

METHOD MR_FirstCycle : BOOL
VAR_INPUT
	sName 			: STRING;
	sFileDir		: STRING(255);
	sFileName		: STRING(255);
	sAmsNetId		: T_AmsNetID;
	bAddTimeStamp	: BOOL;
	bAddHeader		: BOOL;
END_VAR
THIS^.sName := sName;
THIS^.sFileDir := sFileDir;
THIS^.sFileName := sFileName;
THIS^.sAmsNetId := sAmsNetId;
THIS^.bAddTimeStamp := bAddTimeStamp;
THIS^.bAddHeader := bAddHeader;

M_SetNewPath();
END_METHOD

METHOD MR_Init : BOOL
VAR_INPUT
END_VAR
IF eFileLoggerState = FILE_LOGGER_UNINITIALIZED THEN
	bBusy := TRUE;
	MR_Init := FALSE;
	eFileLoggerState := FILE_LOGGER_INITIALIZING;
	
ELSIF eFileLoggerState >= FILE_LOGGER_READY THEN
	bBusy := FALSE;
	MR_Init := TRUE;
	
END_IF
END_METHOD

METHOD MR_Reset : BOOL
IF eFileLoggerState >= FILE_LOGGER_IDLE AND eFileLoggerState <> FILE_LOGGER_METHOD_DONE THEN
	bBusy := TRUE;
	MR_Reset := FALSE;
	eFileLoggerState := FILE_LOGGER_RESET;	

ELSIF eFileLoggerState = FILE_LOGGER_METHOD_DONE THEN
	bBusy := FALSE;
	MR_Reset := TRUE;

END_IF
END_METHOD

METHOD MR_SelectPath : BOOL
VAR_INPUT
	sFileDir								: STRING; 			(* CSV source file directory name *)
	sFileName 								: STRING; 			(* CSV source file name *)
END_VAR
IF eFileLoggerState = FILE_LOGGER_IDLE THEN
	THIS^.sFileDir := sFileDir;	
	THIS^.sFileName := sFileName;	
	bBusy := TRUE;
	MR_SelectPath := FALSE;
	eFileLoggerState := FILE_LOGGER_SELECT_PATH;
	
ELSIF eFileLoggerState = FILE_LOGGER_METHOD_DONE THEN
	bBusy := FALSE;
	MR_SelectPath := TRUE;
	
END_IF
END_METHOD

METHOD PROTECTED MS_Aborting
fbCreateDir( bExecute := FALSE);
fbFileOpen( bExecute := FALSE);
fbFilePuts( bExecute := FALSE);
fbFileClose( bExecute := FALSE);
//fbGetTime( START := FALSE);

FOR iCurrentBufferLine := 1 TO iBUFFER_SIZE BY 1 DO
	MEMSET(ADR(arrMessageBuffer[iCurrentBufferLine]),0,SIZEOF(arrMessageBuffer[iCurrentBufferLine]));
	arrMessageBufferPresence[iCurrentBufferLine] := FALSE;
	
END_FOR

iCurrentBufferLine := 1;
iCurrentBufferLineForFile := 1;

MEMSET(ADR(sTime),0,SIZEOF(sTime));
MEMSET(ADR(sFileDate),0,SIZEOF(sFileDate));
MEMSET(ADR(sLogMessage),0,SIZEOF(sLogMessage));

stTime.wDay 			:= 0;
stTime.wDayOfWeek 		:= 0;
stTime.wHour 			:= 0;
stTime.wMilliseconds 	:= 0;
stTime.wMinute 			:= 0;
stTime.wMonth 			:= 0;
stTime.wSecond 			:= 0;
stTime.wYear 			:= 0;

bActive		:= FALSE;
bBusy 		:= FALSE;
bError 		:= FALSE;
iErrorID 	:= 0;

eFileLoggerInitState := FILE_LOGGER_INIT_GET_TIME;
eFileLoggerAddLogsState := FILE_LOGGER_ADD_LOGS_OPEN;
eFileLoggerState := FILE_LOGGER_UNINITIALIZED;
END_METHOD

METHOD PROTECTED MS_AddLogs
CASE eFileLoggerAddLogsState OF
	FILE_LOGGER_ADD_LOGS_OPEN:
		IF NOT fbFileOpen.bError THEN
			fbFileOpen( sNetId 		:= sAmsNetId,
						sPathName 	:= FUN_MergeStrings4(sStr1 := sFilePath,'_',LEFT(sTime,10),'.txt'),
						bExecute 	:= TRUE,
						tTimeout	:= DEFAULT_ADS_TIMEOUT,
						nMode		:= FOPEN_MODEAPPEND OR FOPEN_MODEPLUS);
							
			IF NOT fbFileOpen.bBusy THEN
				fbFileOpen(bExecute := FALSE);				
				hFile := fbFileOpen.hFile;;
				eFileLoggerAddLogsState := FILE_LOGGER_ADD_LOGS_WRITTE;
			
			END_IF
		ELSE
			fbFileOpen( bExecute := FALSE);
			bError := fbFileOpen.bError;
			iErrorID := fbFileOpen.nErrId;

		END_IF
	

	FILE_LOGGER_ADD_LOGS_WRITTE:
		IF NOT fbFilePuts.bError THEN
			fbFilePuts( sNetId		:= sAmsNetId,
						hFile 		:= hFile,
						sLine 		:= arrMessageBuffer[iCurrentBufferLineForFile],
						bExecute 	:= TRUE,
						tTimeout 	:= DEFAULT_ADS_TIMEOUT);	
					
			IF NOT fbFilePuts.bBusy THEN				
				eFileLoggerAddLogsState := FILE_LOGGER_ADD_LOGS_WRITTE_DONE;
				
			END_IF
			
		ELSE
			fbFilePuts( bExecute := FALSE);
			bError := fbFilePuts.bError;
			iErrorID := fbFilePuts.nErrId;
			
		END_IF	

		
	FILE_LOGGER_ADD_LOGS_WRITTE_DONE:
		fbFilePuts( bExecute := FALSE);	
		iCurrentBufferLineForFile := iCurrentBufferLineForFile + 1;	
		
		IF iCurrentBufferLineForFile >= iBUFFER_SIZE THEN
			iCurrentBufferLineForFile := 1;
		ELSIF iCurrentBufferLineForFile < iCurrentBufferLine THEN
			eFileLoggerAddLogsState := FILE_LOGGER_ADD_LOGS_WRITTE;
		ELSIF iCurrentBufferLineForFile >= iCurrentBufferLine THEN
			eFileLoggerAddLogsState := FILE_LOGGER_ADD_LOGS_CLOSE;
		END_IF;

	
	FILE_LOGGER_ADD_LOGS_CLOSE:
		IF NOT fbFileClose.bError THEN
			fbFileClose(	sNetId := sAmsNetId,
							hFile := hFile,
							bExecute := TRUE,
							tTimeout := DEFAULT_ADS_TIMEOUT);
							
			IF NOT fbFileClose.bBusy THEN
				fbFileClose( bExecute := FALSE);
				eFileLoggerAddLogsState := FILE_LOGGER_ADD_LOGS_OPEN;
				eFileLoggerState := FILE_LOGGER_IDLE;

			END_IF
		ELSE
			bError := fbFileClose.bError;
			iErrorID := fbFileClose.nErrId;
			fbFileClose( bExecute := FALSE);
			
		END_IF
		
END_CASE
END_METHOD

METHOD PROTECTED MS_Idle
VAR_INPUT
END_VAR
IF iCurrentBufferLineForFile < iCurrentBufferLine THEN
	eFileLoggerState := FILE_LOGGER_ADD_LOGS;

END_IF
END_METHOD

METHOD PROTECTED MS_Initializing //C:\TwinCAT\log\filelog.txt
CASE eFileLoggerInitState OF
	FILE_LOGGER_INIT_CREATE_DIR:
		fbCreateDir(sNetId 		:= sAmsNetId,
					sPathName 	:= sFileDir,
					bExecute 	:= TRUE,
					tTimeout 	:= DEFAULT_ADS_TIMEOUT);
					
		IF NOT fbCreateDir.bBusy THEN
			eFileLoggerInitState := FILE_LOGGER_INIT_GET_TIME;
			fbCreateDir( bExecute := FALSE);
			
		END_IF
		
	FILE_LOGGER_INIT_GET_TIME:
		IF fbMachineTime.bValid THEN
			stTime := fbMachineTime.systemTime;
			sTime := SYSTEMTIME_TO_STRING(stTime);
			sFileDate := LEFT(sTime,10);
			eFileLoggerInitState := FILE_LOGGER_INIT_CREATE_FILE;
			
		END_IF
		
	FILE_LOGGER_INIT_CREATE_FILE:
		IF NOT fbFileOpen.bError THEN
			fbFileOpen( sNetId 		:= sAmsNetId,
						sPathName 	:= FUN_MergeStrings4(sFilePath,'_',LEFT(sTime,10),'.txt'),
						bExecute 	:= TRUE,
						tTimeout	:= DEFAULT_ADS_TIMEOUT,
						nMode		:= FOPEN_MODEAPPEND OR FOPEN_MODEPLUS);
							
			IF NOT fbFileOpen.bBusy THEN
				hFile := fbFileOpen.hFile;
				fbFileOpen(bExecute := FALSE);		
				
				IF bAddHeader THEN 
					eFileLoggerInitState := FILE_LOGGER_INIT_ADD_HEADER;
					
				ELSE
					eFileLoggerInitState := FILE_LOGGER_INIT_CLOSE_FILE;
					
				END_IF							
			END_IF
		ELSE
			bError := fbFileOpen.bError;
			iErrorID := fbFileOpen.nErrId;
			fbFileOpen( bExecute := FALSE);
			
		END_IF
		
	FILE_LOGGER_INIT_ADD_HEADER:
	
		IF NOT fbFilePuts.bError THEN
			fbFilePuts(	sNetId := sAmsNetId,
						hFile := hFile,
						sLine := CONCAT('----- Logger file initialized at ',CONCAT(LEFT(sTime,23),' ----- $n')),
						bExecute := TRUE,
						tTimeout := DEFAULT_ADS_TIMEOUT);

			IF NOT fbFilePuts.bBusy THEN
				eFileLoggerInitState := FILE_LOGGER_INIT_CLOSE_FILE;
				fbFilePuts( bExecute := FALSE);
				
			END_IF	
		ELSE
			bError := fbFilePuts.bError;
			iErrorID := fbFilePuts.nErrId;
			fbFilePuts( bExecute := FALSE);
			
		END_IF
	
	FILE_LOGGER_INIT_CLOSE_FILE:
		IF NOT fbFileClose.bError THEN
			fbFileClose( sNetId 		:= sAmsNetId,
							hFile 		:= hFile,
							bExecute 	:= TRUE,
							tTimeout 	:= DEFAULT_ADS_TIMEOUT);
							
			IF NOT fbFileClose.bBusy THEN
				eFileLoggerInitState := FILE_LOGGER_INIT_DONE;
				fbFileClose( bExecute := FALSE);
				
			END_IF
		ELSE
			bError := fbFileClose.bError;
			iErrorID := fbFileClose.nErrId;
			fbFileClose( bExecute := FALSE);
			
		END_IF
	
	FILE_LOGGER_INIT_DONE:
		eFileLoggerInitState := FILE_LOGGER_INIT_CREATE_DIR;
		eFileLoggerState := FILE_LOGGER_IDLE;
		
END_CASE
END_METHOD

METHOD PROTECTED MS_MethodDone
VAR_INPUT
END_VAR
IF NOT bBusy THEN
	eFileLoggerState := FILE_LOGGER_IDLE;

END_IF
END_METHOD

METHOD PROTECTED MS_Ready
VAR_INPUT
END_VAR
eFileLoggerState := FILE_LOGGER_IDLE;
END_METHOD

METHOD PROTECTED MS_Reset
VAR_INPUT
END_VAR
IF M_ResetParameters() THEN
	eFileLoggerState := FILE_LOGGER_METHOD_DONE;
	
END_IF
END_METHOD

METHOD MS_SelectPath : BOOL
VAR_INPUT
END_VAR
IF M_SetNewPath() THEN
	eFileLoggerState := FILE_LOGGER_METHOD_DONE;
	
END_IF
END_METHOD

METHOD PROTECTED MS_Uninitialized
;
END_METHOD

PROPERTY Name : STRING
GET
Name := sName;
END_GET
SET
sName := Name;
END_SET
END_PROPERTY

METHOD PROTECTED StateMachine
CASE eFileLoggerState OF
	FILE_LOGGER_UNINITIALIZED:
		MS_Uninitialized();
		
	FILE_LOGGER_INITIALIZING:
		MS_Initializing();
		
	FILE_LOGGER_IDLE:
		MS_Idle();
		
	FILE_LOGGER_ADD_LOGS:
		MS_AddLogs();	
		
	FILE_LOGGER_RESET:
		MS_Reset();
		
	FILE_LOGGER_METHOD_DONE:
		MS_MethodDone();
	
	FILE_LOGGER_ABORTING:
		MS_Aborting();
	
END_CASE
END_METHOD

END_FUNCTION_BLOCK

// ---- POUs/Libs/Utilities/StringMerge/FUN_MergeStrings6.TcPOU
(* 
:Description: This function is used to merge 6 strings
*)
FUNCTION FUN_MergeStrings6 : STRING(300)
VAR_INPUT
	sStr1	: STRING;		(* First string in merge row *)
	sStr2	: STRING;		(* Second string in merge row *)
	sStr3	: STRING;		(* Third string in merge row *)
	sStr4	: STRING;		(* Fourth string in merge row *)
	sStr5	: STRING;		(* Fifth string in merge row *)
	sStr6	: STRING;		(* Sixth string in merge row *)
END_VAR

FUN_MergeStrings6 := CONCAT(sStr1,sStr2);
FUN_MergeStrings6 := CONCAT(FUN_MergeStrings6, sStr3);
FUN_MergeStrings6 := CONCAT(FUN_MergeStrings6, sStr4);
FUN_MergeStrings6 := CONCAT(FUN_MergeStrings6, sStr5);
FUN_MergeStrings6 := CONCAT(FUN_MergeStrings6, sStr6);

END_FUNCTION

// ---- POUs/Libs/Utilities/StringMerge/FUN_MergeStrings4.TcPOU
(* 
:Description: This function is used to merge 5 strings
*)
FUNCTION FUN_MergeStrings4 : STRING
VAR_INPUT
	sStr1	: STRING;			(* Fifth string in merge row *)
	sStr2	: STRING;			(* Fourth string in merge row *)
	sStr3	: STRING;			(* Fourth string in merge row *)
	sStr4	: STRING;			(* Fourth string in merge row *)

END_VAR

FUN_MergeStrings4 := CONCAT(sStr1,sStr2);
FUN_MergeStrings4 := CONCAT(FUN_MergeStrings4,sStr3);
FUN_MergeStrings4 := CONCAT(FUN_MergeStrings4,sStr4);

END_FUNCTION

// ---- POUs/Machine/Recipes Manager/PRG_RecipesManager.TcPOU
PROGRAM PRG_RecipesManager
VAR CONSTANT
	sDEFAULT_STORAGE_PATH		: STRING(512) := 'C:\TwinCAT\Tests\Recipes\';	(* Default storage path for recipe files *)
	sDEFAULT_RECIPE_DEFINITION	: STRING := 'Recipes';						(* Default definition of Recipe configuration from RecipesManager *)
	sDEFAULT_RECIPE_NAME		: STRING := 'R1';							(* Default name of selected Recipe *)
END_VAR
VAR		
	bFirstCycle 		: BOOL := TRUE;
	sTest1 				: REFERENCE TO STRING;
	fbRecipesControler	: FB_RecipesControler;	(* Recipes Controler *)
END_VAR

IF bFirstCycle AND fbRecipesControler.RecipeValuesAdrAvailable THEN
	bFirstCycle := FALSE;
	fbRecipesControler.MR_FirstCycle(	sLocalStoragePath 	:= sDEFAULT_STORAGE_PATH,
										sRecipesDefinition	:= sDEFAULT_RECIPE_DEFINITION,
										sDefaultRecipeName	:= sDEFAULT_RECIPE_NAME);					
	
	(* Assign recipe parameters *)								
	stShell.stRecipeData.rpVar1.MR_FirstCycle(	eType := VISU_CTRL_RECIPES_PARAMETER_TYPE_REAL, 
												sName := 'Var1', 
												pFileValueAdr := fbRecipesControler.RecipeValuesAdr[0]);
										
	stShell.stRecipeData.rpVar2.MR_FirstCycle(	eType := VISU_CTRL_RECIPES_PARAMETER_TYPE_REAL, 
												sName := 'Var2', 
												pFileValueAdr := fbRecipesControler.RecipeValuesAdr[1]);
												
	stShell.stRecipeData.rpVar3.MR_FirstCycle(	eType := VISU_CTRL_RECIPES_PARAMETER_TYPE_REAL, 
												sName := 'Var3', 
												pFileValueAdr := fbRecipesControler.RecipeValuesAdr[2]);
												
	stShell.stRecipeData.rpVar4.MR_FirstCycle(	eType := VISU_CTRL_RECIPES_PARAMETER_TYPE_INT, 
												sName := 'Var4', 
												pFileValueAdr := fbRecipesControler.RecipeValuesAdr[3]);			
												
	stShell.stRecipeData.rpVar5.MR_FirstCycle(	eType := VISU_CTRL_RECIPES_PARAMETER_TYPE_INT, 
												sName := 'Var5', 
												pFileValueAdr := fbRecipesControler.RecipeValuesAdr[4]);
												
	stShell.stRecipeData.rpVar6.MR_FirstCycle(	eType := VISU_CTRL_RECIPES_PARAMETER_TYPE_INT, 
												sName := 'Var6', 
												pFileValueAdr := fbRecipesControler.RecipeValuesAdr[5]);
												
	stShell.stRecipeData.rpVar7.MR_FirstCycle(	eType := VISU_CTRL_RECIPES_PARAMETER_TYPE_STRING, 
												sName := 'Var7', 
												pFileValueAdr := fbRecipesControler.RecipeValuesAdr[6]);
												
	stShell.stRecipeData.rpVar8.MR_FirstCycle(	eType := VISU_CTRL_RECIPES_PARAMETER_TYPE_STRING, 
												sName := 'Var8', 
												pFileValueAdr := fbRecipesControler.RecipeValuesAdr[7]);
												
	stShell.stRecipeData.rpVar9.MR_FirstCycle(	eType := VISU_CTRL_RECIPES_PARAMETER_TYPE_STRING, 
												sName := 'Var9', 
												pFileValueAdr := fbRecipesControler.RecipeValuesAdr[8]);
												
	stShell.stRecipeData.rpVar10.MR_FirstCycle(	eType := VISU_CTRL_RECIPES_PARAMETER_TYPE_BOOL, 
												sName := 'Var10', 
												pFileValueAdr := fbRecipesControler.RecipeValuesAdr[9]);
	
	(* Assign recipes controler reference to Shell API*)
	stShell.stPlatform.ref_fbRecipesManager REF= fbRecipesControler;
	
	(* Set assignamnet done bit for visu controler *)
	stShell.stFlags.bRecipesCtrlAssignamentsDone := TRUE;
END_IF

fbRecipesControler();

END_PROGRAM

// ---- POUs/Libs/Utilities/Recipes Manager/FB_RecipesControler.TcPOU
(* 
:Description: This function block is used to control the recipe manager feature
*) 
FUNCTION_BLOCK FB_RecipesControler IMPLEMENTS I_RecipesManager
VAR	
	bFirstCycle: BOOL := TRUE;
	iLoop : INT;
	
	(* Internal commands *)
	bInit						: BOOL;									(*  *)
	bAbort						: BOOL;									(*  *)
	bCreate						: BOOL;									(*  *)
	bLoad						: BOOL;									(*  *)
	bLoadAndWrite				: BOOL;									(*  *)
	bRead						: BOOL;									(*  *)
	bReadAndSave				: BOOL;									(*  *)
	bRemove						: BOOL;									(*  *)
	bSave						: BOOL;									(*  *)
	bWrite						: BOOL;									(*  *)
	bGetRecipeCount				: BOOL;									(*  *)
	bGetNameArray				: BOOL;									(*  *)
	bGetVariableNames			: BOOL;									(*  *)
	bGetRecipeNames				: BOOL;									(*  *)
	bGetVariableValues			: BOOL;									(*  *)
	bReload						: BOOL;									(*  *)
	bRestore					: BOOL;									(*  *)
	bBackup						: BOOL;									(*  *)
	
	(* Internal parameters *)
	sStoragePath				: STRING;
	sLocalStoragePath			: STRING;								(*  *)
	sBackupStoragePath			: STRING;
	sRecipesDefinition			: STRING;								(*  *)
	sRecipeName					: STRING;								(*  *)
	
	(* Internal status *)
	bActive						: BOOL;									(*  *)
	bBusy						: BOOL;									(*  *)
	bError						: BOOL;									(*  *)
	iErrorId 					: DWORD;								(*  *)
	
	eStateMachine				: E_RecipesManagerState;				(*  *)
	eStateMachineInit			: E_RecipesmanagerStateInit;			(*  *)
	eStateMachineReload			: E_RecipesManagerStateReload;
	eStateMachineCreateRemove	: E_RecipesManagerStateCreateRemove;	(*  *)
	eStateMachineBackup			: E_RecipesManagerStateBackup;	(*  *)
	
	bLastSetStoragePathResult	: BOOL;									(*  *)
	iLastResult					: DWORD;								(*  *)
	eLastResult					: E_RecipesManagerReturns;				(*  *)
	
	iRecipesCount				: USINT;
	arrVariableNames			: ARRAY [0..iMAX_NUMBER_OF_VARIABLES_IN_RECIPES-1] OF STRING;
	arrRecipesNames				: ARRAY	[0..iMAX_NUMBER_OF_RECIPES-1] OF STRING;
	arrRecipeValues				: ARRAY [0..iMAX_NUMBER_OF_VARIABLES_IN_RECIPES-1] OF STRING;
	
	//iArrRecipeValuesAdr			: PVOID := ADR(arrRecipeValues);
	arrRecipeValuesAdr			: ARRAY [0..iMAX_NUMBER_OF_VARIABLES_IN_RECIPES-1] OF PVOID;
	bRecipeFileValuesAdrAvailable	: BOOL := FALSE;
	
	(* Function blocks *)
	fbRecipeManager 			: RecipeManCommands; (* Recipes manager clontroling FB *)
	
	(* Tc3 EventLogger - messages *)
	bAlarmFailed			: FB_TcAlarm;				(*  *)	
	fbAlarmParameter		: FB_TcAlarm;				(*  *)
	fbAlarmNotInitialized	: FB_TcAlarm;				(*  *)
	fbAlarmNotImplemented	: FB_TcAlarm;				(*  *)
	fbAlarmNoObject			: FB_TcAlarm;				(*  *)
	fbAlarmFileNoMemory		: FB_TcAlarm;				(*  *)
	fbAlarmFileNotFound		: FB_TcAlarm;				(*  *)
	fbAlarmRecipeMismatch	: FB_TcAlarm;				(*  *)
	fbAlarmRecipeSave		: FB_TcAlarm;				(*  *)
	fbAlarmRecipeNotFound	: FB_TcAlarm;				(*  *)
	fbAlarmDefNotFound		: FB_TcAlarm;				(*  *)
	fbAlarmAlreadyExist		: FB_TcAlarm;				(*  *)
	fbAlarmNoManagerSet		: FB_TcAlarm;				(*  *)
	fbAlarmNotAllVariable	: FB_TcAlarm;				(*  *)
	fbAlarmRecipeNoMemory	: FB_TcAlarm;				(*  *)
	fbAlarmManagerLocked	: FB_TcAlarm;				(*  *)
	fbAlarmSourceExhausted	: FB_TcAlarm;				(*  *)
	fbAlarmTargetExhausted	: FB_TcAlarm;				(*  *)
	fbAlarmSourceIllegal	: FB_TcAlarm;				(*  *)
	
	
	rtError		: R_TRIG; 					(* Rising edge trigger for function block error *)
END_VAR
(*
Version history:

+-------------+------------+----------------+----------+----------------------------------------------------------------+
|Date         | Version    | created under  | Author   | Remark                                                         |
+=============+============+================+==========+================================================================+
|2021-11      | 1.0.0.0    | V3.1.4024.22   | ADBO     | Function block created                                         |
+-------------+------------+----------------+----------+----------------------------------------------------------------+
|2022-06      | 1.0.1.0    | V3.1.4024.22   | ADBO     | Fixes for all detected bugs after tests with Visu controler    |
+-------------+------------+----------------+----------+----------------------------------------------------------------+

*)

IF bFirstCycle THEN
	bFirstCycle := FALSE;
	
	FOR iLoop := 0 TO iMAX_NUMBER_OF_VARIABLES_IN_RECIPES-1 DO
		arrRecipeValuesAdr[iLoop] := ADR(arrRecipeValues[iLoop]);
	END_FOR
	
	bRecipeFileValuesAdrAvailable := TRUE;
	
	bAlarmFailed.CreateEx( stEventEntry := TC_EVENTS.ShellRecipesEventClass.Failed, 
									bWithConfirmation := 1,
									ipSourceInfo := 0);
		
	fbAlarmParameter.CreateEx( stEventEntry := TC_EVENTS.ShellRecipesEventClass.Parameter, 
									bWithConfirmation := 1,
									ipSourceInfo := 0);
									
	fbAlarmNotInitialized.CreateEx( stEventEntry := TC_EVENTS.ShellRecipesEventClass.NotInitialized, 
									bWithConfirmation := 1,
									ipSourceInfo := 0);		
									
	fbAlarmNotImplemented.CreateEx( stEventEntry := TC_EVENTS.ShellRecipesEventClass.NotImplemented, 
									bWithConfirmation := 1,
									ipSourceInfo := 0);
		
	fbAlarmNoObject.CreateEx( stEventEntry := TC_EVENTS.ShellRecipesEventClass.NoObject, 
									bWithConfirmation := 1,
									ipSourceInfo := 0);
									
	fbAlarmFileNoMemory.CreateEx( stEventEntry := TC_EVENTS.ShellRecipesEventClass.FileNoMemory, 
									bWithConfirmation := 1,
									ipSourceInfo := 0);	
									
	fbAlarmFileNotFound.CreateEx( stEventEntry := TC_EVENTS.ShellRecipesEventClass.FileNotFound, 
									bWithConfirmation := 1,
									ipSourceInfo := 0);
		
	fbAlarmRecipeMismatch.CreateEx( stEventEntry := TC_EVENTS.ShellRecipesEventClass.RecipeMismatch, 
									bWithConfirmation := 1,
									ipSourceInfo := 0);
									
	fbAlarmRecipeSave.CreateEx( stEventEntry := TC_EVENTS.ShellRecipesEventClass.RecipeSave, 
									bWithConfirmation := 1,
									ipSourceInfo := 0);	

	fbAlarmRecipeNotFound.CreateEx( stEventEntry := TC_EVENTS.ShellRecipesEventClass.RecipeNotFound, 
									bWithConfirmation := 1,
									ipSourceInfo := 0);
		
	fbAlarmDefNotFound.CreateEx( stEventEntry := TC_EVENTS.ShellRecipesEventClass.DefNotFound, 
									bWithConfirmation := 1,
									ipSourceInfo := 0);
									
	fbAlarmAlreadyExist.CreateEx( stEventEntry := TC_EVENTS.ShellRecipesEventClass.AlreadyExist, 
									bWithConfirmation := 1,
									ipSourceInfo := 0);	
									
	fbAlarmNoManagerSet.CreateEx( stEventEntry := TC_EVENTS.ShellRecipesEventClass.NoManagerSet, 
									bWithConfirmation := 1,
									ipSourceInfo := 0);
		
	fbAlarmNotAllVariable.CreateEx( stEventEntry := TC_EVENTS.ShellRecipesEventClass.NotAllVariable, 
									bWithConfirmation := 1,
									ipSourceInfo := 0);
									
	fbAlarmRecipeNoMemory.CreateEx( stEventEntry := TC_EVENTS.ShellRecipesEventClass.RecipeNoMemory, 
									bWithConfirmation := 1,
									ipSourceInfo := 0);	
									
	fbAlarmManagerLocked.CreateEx( stEventEntry := TC_EVENTS.ShellRecipesEventClass.ManagerLocked, 
									bWithConfirmation := 1,
									ipSourceInfo := 0);
		
	fbAlarmSourceExhausted.CreateEx( stEventEntry := TC_EVENTS.ShellRecipesEventClass.SourceExhausted, 
									bWithConfirmation := 1,
									ipSourceInfo := 0);
									
	fbAlarmTargetExhausted.CreateEx( stEventEntry := TC_EVENTS.ShellRecipesEventClass.TargetExhausted, 
									bWithConfirmation := 1,
									ipSourceInfo := 0);	

	fbAlarmSourceIllegal.CreateEx( stEventEntry := TC_EVENTS.ShellRecipesEventClass.SourceIllegal, 
									bWithConfirmation := 1,
									ipSourceInfo := 0);
							
END_IF

(* Control active flag *)
bActive := eStateMachine >= RECIPES_MANAGER_IDLE;

(* Set last result enum*)
CASE iLastResult OF
	ERR_OK:
		eLastResult := RECIPES_MANAGER_ERR_OK;
		
	ERR_FAILED:
		eLastResult := RECIPES_MANAGER_ERR_FAILED;
		bAlarmFailed.Raise(0);
		
	ERR_PARAMETER:
		eLastResult := RECIPES_MANAGER_ERR_PARAMETER;
		fbAlarmParameter.Raise(0);
		
	ERR_NOTINITIALIZED:
		eLastResult := RECIPES_MANAGER_ERR_NOTINITALIZED;
		fbAlarmNotInitialized.Raise(0);
		
	ERR_NOTIMPLEMENTED:
		eLastResult := RECIPES_MANAGER_ERR_NOIMPLEMENTED;
		fbAlarmNotImplemented.Raise(0);
		
	ERR_NO_OBJECT:
		eLastResult := RECIPES_MANAGER_ERR_NO_OBJECT;
		fbAlarmNoObject.Raise(0);
		
	ERR_NOMEMORY:
		eLastResult := RECIPES_MANAGER_ERR_NOMEMORY;
		fbAlarmFileNoMemory.Raise(0);
		
	ERR_RECIPE_FILE_NOT_FOUND:
		eLastResult := RECIPES_MANAGER_ERR_RECIPE_FILE_NOT_FOUND;
		fbAlarmFileNotFound.Raise(0);
		
	ERR_RECIPE_MISMATCH:
		eLastResult := RECIPES_MANAGER_ERR_RECIPE_MISMATCH;
		fbAlarmRecipeMismatch.Raise(0);
		
	ERR_RECIPE_SAVE_ERR:
		eLastResult := RECIPES_MANAGER_ERR_RECIPE_SAVE_ERR;
		fbAlarmRecipeSave.Raise(0);
		
	ERR_RECIPE_NOT_FOUND:
		eLastResult := RECIPES_MANAGER_ERR_RECIPE_NOT_FOUND;
		fbAlarmRecipeNotFound.Raise(0);
		
	ERR_RECIPE_DEFINITION_NOT_FOUND:
		eLastResult := RECIPES_MANAGER_ERR_RECIPE_DEFINITION_NOT_FOUND;
		fbAlarmDefNotFound.Raise(0);
		
	ERR_RECIPE_ALREADY_EXIST:
		eLastResult := RECIPES_MANAGER_ERR_RECIPE_ALREADY_EXIST;
		fbAlarmAlreadyExist.Raise(0);
		
	ERR_NO_RECIPE_MANAGER_SET:
		eLastResult := RECIPES_MANAGER_ERR_NO_RECIPE_MANAGER_SET;
		fbAlarmNoManagerSet.Raise(0);
		
	ERR_RECIPE_NOT_ALL_VARIABLES_WERE_LOADED:
		eLastResult := RECIPES_MANAGER_ERR_RECIPE_NOT_ALL_VARIABLES_WERE_LOADED;
		fbAlarmNotAllVariable.Raise(0);
		
	ERR_RECIPE_NOMEMORY:
		eLastResult := RECIPES_MANAGER_ERR_NOMEMORY;
		fbAlarmRecipeNoMemory.Raise(0);
		
	ERR_RECIPE_MANAGER_LOCKED_DURING_ONLINE_CHANGE:
		eLastResult := RECIPES_MANAGER_ERR_RECIPES_MANAGER_LOCKED;
		fbAlarmManagerLocked.Raise(0);
		
	ERR_SOURCE_EXHAUSTED:
		eLastResult := RECIPES_MANAGER_ERR_SOURCE_EXHAUSTED;
		fbAlarmSourceExhausted.Raise(0);
		
	ERR_TARGET_EXHAUSTED:
		eLastResult := RECIPES_MANAGER_ERR_TARGET_EXHAUSTED;
		fbAlarmTargetExhausted.Raise(0);
		
	ERR_SOURCE_ILLEGAL:
		eLastResult := RECIPES_MANAGER_ERR_SOURCE_ILLEGAL;
		fbAlarmSourceIllegal.Raise(0);
		
END_CASE

(* Report errors that occur *)
rtError(CLK:=bError);

IF rtError.Q THEN 
	fbMachineLogger.MR_AddLogs(FUN_MergeStrings5('Recipes_Manager', ' : Error occured (error ID: ', UDINT_TO_STRING(iErrorID), ')', ''));
END_IF

(* Run state machine *)
StateMachine();

(* Execute recipe manager instance *)
fbRecipeManager();

PROPERTY Active : REFERENCE TO BOOL
GET
Active REF= bActive;
END_GET
END_PROPERTY

PROPERTY Busy : REFERENCE TO BOOL
GET
Busy REF= bBusy;
END_GET
END_PROPERTY

PROPERTY Error : REFERENCE TO BOOL
GET
Error REF= bError;
END_GET
END_PROPERTY

PROPERTY ErrorID : REFERENCE TO DWORD
GET
ErrorID REF= iErrorId;
END_GET
END_PROPERTY

PROPERTY LastResult : REFERENCE TO E_RecipesManagerReturns
GET
LastResult REF= eLastResult;
END_GET
END_PROPERTY

METHOD PRIVATE M_GetRecipesCount
VAR_INPUT
END_VAR
iRecipesCount := INT_TO_USINT(fbRecipeManager.GetRecipeCount(sRecipesDefinition));
iLastResult := fbRecipeManager.GetLastError();
END_METHOD

METHOD M_GetRecipesNames : BOOL
VAR
	i : USINT;
END_VAR
//FOR i := 0 TO iMAX_NUMBER_OF_RECIPES-1 DO
	iLastResult := fbRecipeManager.GetRecipeNames( 	RecipeDefinitionName	:= sRecipesDefinition,
													pStrings				:= ADR(arrRecipesNames),
													iSize 					:= iMAX_RECIPE_NAME_LENGTH,
													iStartIndex 			:= 0);
//END_FOR
END_METHOD

METHOD PRIVATE M_GetVariableNames
VAR
	i : USINT;
END_VAR
//FOR i := 0 TO iMAX_NUMBER_OF_VARIABLES_IN_RECIPES-1 DO
	iLastResult := fbRecipeManager.GetRecipeVariableNames(	RecipeDefinitionName	:= sRecipesDefinition,
															RecipeName				:= sRecipeName,
															pStrings 				:= ADR(arrVariableNames),
															iSize 					:= iMAX_NUMBER_OF_VARIABLES_IN_RECIPES,
															iStartIndex				:= 0);
//END_FOR
END_METHOD

METHOD PRIVATE M_GetVariableValues
VAR
	i : USINT;
END_VAR
//FOR i := 0 TO iMAX_NUMBER_OF_VARIABLES_IN_RECIPES-1 DO
iLastResult := fbRecipeManager.GetRecipeValues( RecipeDefinitionName 	:= sRecipesDefinition,
												RecipeName 				:= sRecipeName,
												pStrings 				:= ADR(arrRecipeValues),
												iSize 					:= iMAX_NUMBER_OF_VARIABLES_IN_RECIPES,
												iStartIndex 			:= 0,
												iStringLength 			:= 80);//255);
//	IF iLastResult <> ERR_OK THEN
//		EXIT;
//	END_IF
//END_FOR
END_METHOD

METHOD PRIVATE M_ReloadRecipes
VAR_INPUT
END_VAR
iLastResult := fbRecipeManager.ReloadRecipes(sRecipesDefinition);
END_METHOD

METHOD PRIVATE M_SetStoragePath
bLastSetStoragePathResult := fbRecipeManager.SetStoragePath(sStoragePath);
END_METHOD

METHOD MR_Abort : BOOL
VAR_INPUT
END_VAR
IF eStateMachine >= RECIPES_MANAGER_INITIALIZATION THEN
	bAbort := TRUE;
	bBusy := TRUE;
	eStateMachine := RECIPES_MANAGER_ABORTING;
	fbMachineLogger.MR_AddLogs(CONCAT('Recipes_Manager',' : abort requested'));	
	
ELSIF eStateMachine = RECIPES_MANAGER_UNINITIALIZED THEN
	bAbort := FALSE;
	bBusy := FALSE;
	MR_Abort := TRUE;
	fbMachineLogger.MR_AddLogs(CONCAT('Recipes_Manager',' : abort done'));	
	
END_IF
END_METHOD

METHOD MR_Backup : BOOL
VAR_INPUT
	sRecipesDefinition		: STRING;
	sRecipeName				: STRING;
	sBackupStoragePath		: STRING;
END_VAR
IF eStateMachine = RECIPES_MANAGER_IDLE THEN
	bBackup := TRUE;
	bBusy := TRUE;
	bError := FALSE;
	iErrorId := 0;
	THIS^.sRecipesDefinition := sRecipesDefinition;
	THIS^.sRecipeName := sRecipeName;
	THIS^.sBackupStoragePath := sBackupStoragePath;
	sStoragePath := sBackupStoragePath;
	M_SetStoragePath();
	M_ReloadRecipes();
	MR_Backup := FALSE;
	eStateMachine := RECIPES_MANAGER_BACKUP;
	fbMachineLogger.MR_AddLogs(CONCAT('Recipes_Manager',' : recipe backup requested'));	
	
ELSIF eStateMachine = RECIPES_MANAGER_BACKUP_DONE THEN
	sStoragePath := sLocalStoragePath;
	M_SetStoragePath();
	bBackup := FALSE;
	bBusy := FALSE;
	MR_Backup := TRUE;
	fbMachineLogger.MR_AddLogs(CONCAT('Recipes_Manager',' : recipe backup done'));	
	
END_IF
END_METHOD

METHOD MR_Create : BOOL
VAR_INPUT
	sRecipesDefinition : STRING;
	sRecipeName : STRING;
END_VAR
IF eStateMachine = RECIPES_MANAGER_IDLE THEN
	bCreate := TRUE;
	bBusy := TRUE;
	bError := FALSE;
	iErrorId := 0;
	THIS^.sRecipesDefinition := sRecipesDefinition;
	THIS^.sRecipeName := sRecipeName;
	M_ReloadRecipes();
	eStateMachine := RECIPES_MANAGER_CREATE;
	fbMachineLogger.MR_AddLogs(CONCAT('Recipes_Manager',' : recipe creation requested'));		
	
ELSIF eStateMachine = RECIPES_MANAGER_CREATE_DONE THEN
	bCreate := FALSE;
	bBusy := FALSE;
	MR_Create := TRUE;
	fbMachineLogger.MR_AddLogs(CONCAT('Recipes_Manager',' : recipe creation done'));	
	
END_IF
END_METHOD

METHOD MR_FirstCycle : BOOL
VAR_INPUT
	sLocalStoragePath	: STRING;	(* Path where all recipes are stored *)
	sRecipesDefinition	: STRING;	(* Template of recipe defined in RecipeManager - IDE *)
	sDefaultRecipeName	: STRING;	(* Default recipes loaded after start *)
END_VAR
THIS^.sLocalStoragePath := sLocalStoragePath;
THIS^.sRecipesDefinition := sRecipesDefinition;
THIS^.sRecipeName := sDefaultRecipeName;
END_METHOD

METHOD MR_GetRecipesNames : BOOL
VAR_INPUT
	sRecipesDefinition : STRING;
END_VAR
IF eStateMachine = RECIPES_MANAGER_IDLE THEN
	bGetNameArray := TRUE;
	bBusy := TRUE;
	bError := FALSE;
	iErrorId := 0;
	THIS^.sRecipesDefinition := sRecipesDefinition;
	eStateMachine := RECIPES_MANAGER_GET_RECIPE_NAME_ARRAY;
	fbMachineLogger.MR_AddLogs(CONCAT('Recipes_Manager',' : get receipe name requested'));	
	
ELSIF eStateMachine = RECIPES_MANAGER_GET_RECIPE_NAME_ARRAY_DONE THEN
	bGetNameArray := FALSE;
	bBusy := FALSE;
	MR_GetRecipesNames := TRUE;
	fbMachineLogger.MR_AddLogs(CONCAT('Recipes_Manager',' : get receipe name done'));	
	
END_IF
END_METHOD

METHOD MR_GetVariablesNames : BOOL
VAR_INPUT
	sRecipesDefinition	: STRING;
	sRecipeName : STRING;
END_VAR
IF eStateMachine = RECIPES_MANAGER_IDLE THEN
	bGetVariableNames := TRUE;
	bBusy := TRUE;
	bError := FALSE;
	iErrorId := 0;
	THIS^.sRecipesDefinition := sRecipesDefinition;
	THIS^.sRecipeName := sRecipeName;
	eStateMachine := RECIPES_MANAGER_GET_RECIPE_VARIABLE_NAMES;
	fbMachineLogger.MR_AddLogs(CONCAT('Recipes_Manager',' : get variable name requested'));	
	
ELSIF eStateMachine = RECIPES_MANAGER_GET_RECIPE_VARIABLE_NAMES_DONE THEN
	bGetNameArray := FALSE;
	bBusy := FALSE;
	MR_GetVariablesNames := TRUE;
	fbMachineLogger.MR_AddLogs(CONCAT('Recipes_Manager',' : get variable name done'));	
	
END_IF
END_METHOD

METHOD MR_GetVariableValues : BOOL
VAR_INPUT
	sRecipesDefinition	: STRING;
	sRecipeName : STRING;
END_VAR
IF eStateMachine = RECIPES_MANAGER_IDLE THEN
	bGetVariableValues := TRUE;
	bBusy := TRUE;
	bError := FALSE;
	iErrorId := 0;
	THIS^.sRecipesDefinition := sRecipesDefinition;
	THIS^.sRecipeName := sRecipeName;
	eStateMachine := RECIPES_MANAGER_GET_RECIPE_VARIABLE_VALUES;
	fbMachineLogger.MR_AddLogs(CONCAT('Recipes_Manager',' : get variable value requested'));	
	
ELSIF eStateMachine = RECIPES_MANAGER_GET_RECIPE_VARIABLE_VALUES_DONE THEN
	bGetVariableValues := FALSE;
	bBusy := FALSE;
	MR_GetVariableValues := TRUE;
	fbMachineLogger.MR_AddLogs(CONCAT('Recipes_Manager',' : get variable value done'));	
	
END_IF
END_METHOD

METHOD MR_Init : BOOL
VAR_INPUT
END_VAR
IF eStateMachine = RECIPES_MANAGER_UNINITIALIZED THEN
	bInit := TRUE;
	fbMachineLogger.MR_AddLogs(CONCAT('Recipes_Manager',' : initialization requested'));	
	bBusy := TRUE;
	bError := FALSE;
	iErrorId := 0;
	eStateMachineInit := RECIPES_MANAGER_INIT_SET_STORAGE_PATH;
	eStateMachine := RECIPES_MANAGER_INITIALIZATION;
	
//ELSIF eStateMachine = RECIPES_MANAGER_INITIALIZATION AND eStateMachineInit = RECIPES_MANAGER_INIT_DONE THEN
ELSIF eStateMachine = RECIPES_MANAGER_IDLE AND bInit THEN
	bInit := FALSE;	
	bBusy := FALSE;
	MR_Init := TRUE;
	fbMachineLogger.MR_AddLogs(CONCAT('Recipes_Manager',' : initialization done'));	
	
END_IF
END_METHOD

METHOD MR_Load : BOOL
VAR_INPUT
	sRecipesDefinition : STRING;
	sRecipeName : STRING;
END_VAR
IF eStateMachine = RECIPES_MANAGER_IDLE THEN
	bLoad := TRUE;
	bBusy := TRUE;
	bError := FALSE;
	iErrorId := 0;
	THIS^.sRecipesDefinition := sRecipesDefinition;
	THIS^.sRecipeName := sRecipeName;
	M_ReloadRecipes();
	eStateMachine := RECIPES_MANAGER_LOAD;
	fbMachineLogger.MR_AddLogs(CONCAT('Recipes_Manager',' : recipe load requested'));	
	
ELSIF eStateMachine = RECIPES_MANAGER_LOAD_DONE THEN
	bLoad := FALSE;
	bBusy := FALSE;
	MR_Load := TRUE;
	fbMachineLogger.MR_AddLogs(CONCAT('Recipes_Manager',' : recipe load done'));	
	
END_IF
END_METHOD

METHOD MR_LoadAndWritte : BOOL
VAR_INPUT
	sRecipesDefinition : STRING;
	sRecipeName : STRING;
END_VAR
IF eStateMachine = RECIPES_MANAGER_IDLE THEN
	bLoadAndWrite := TRUE;
	bBusy := TRUE;
	bError := FALSE;
	iErrorId := 0;
	THIS^.sRecipesDefinition := sRecipesDefinition;
	THIS^.sRecipeName := sRecipeName;
	M_ReloadRecipes();
	eStateMachine := RECIPES_MANAGER_LOAD_AND_WRITE;
	fbMachineLogger.MR_AddLogs(CONCAT('Recipes_Manager',' : recipe loading and writing requested'));	
	
ELSIF eStateMachine = RECIPES_MANAGER_LOAD_AND_WRITE_DONE THEN
	bLoadAndWrite := FALSE;
	bBusy := FALSE;
	MR_LoadAndWritte := TRUE;
	fbMachineLogger.MR_AddLogs(CONCAT('Recipes_Manager',' : recipe loading and writing done'));	
	
END_IF
END_METHOD

(*
When the command is executed, TwinCAT overwrites the values of the selected recipe with the values read from the controller.
In the process, the values are implicitly stored (in a file on the controller) and simultaneously displayed in the table of the recipe definition.
*)
METHOD MR_Read : BOOL
VAR_INPUT
	sRecipesDefinition : STRING;
	sRecipeName : STRING;
END_VAR
IF eStateMachine = RECIPES_MANAGER_IDLE THEN
	bRead := TRUE;
	bBusy := TRUE;
	bError := FALSE;
	iErrorId := 0;
	THIS^.sRecipesDefinition := sRecipesDefinition;
	THIS^.sRecipeName := sRecipeName;
	M_ReloadRecipes();
	eStateMachine := RECIPES_MANAGER_READ;
	fbMachineLogger.MR_AddLogs(CONCAT('Recipes_Manager',' : recipe read requested'));	
	
ELSIF eStateMachine = RECIPES_MANAGER_READ_DONE THEN
	bRead := FALSE;
	bBusy := FALSE;
	MR_Read := TRUE;
	fbMachineLogger.MR_AddLogs(CONCAT('Recipes_Manager',' : recipe read done'));	
	
END_IF
END_METHOD

METHOD MR_ReadAndSave : BOOL
VAR_INPUT
	sRecipesDefinition : STRING;
	sRecipeName : STRING;
END_VAR
IF eStateMachine = RECIPES_MANAGER_IDLE THEN
	bReadAndSave := TRUE;
	bBusy := TRUE;
	bError := FALSE;
	iErrorId := 0;
	THIS^.sRecipesDefinition := sRecipesDefinition;
	THIS^.sRecipeName := sRecipeName;
	M_ReloadRecipes();
	eStateMachine := RECIPES_MANAGER_READ_AND_SAVE;
	fbMachineLogger.MR_AddLogs(CONCAT('Recipes_Manager',' : recipe read and save requested'));		
	
ELSIF eStateMachine = RECIPES_MANAGER_READ_AND_SAVE_DONE THEN
	bReadAndSave := FALSE;
	bBusy := FALSE;
	MR_ReadAndSave := TRUE;
	fbMachineLogger.MR_AddLogs(CONCAT('Recipes_Manager',' : recipe read and save done'));
	
END_IF
END_METHOD

METHOD MR_Reload : BOOL
VAR_INPUT
	sRecipeName : STRING;
	sRecipesDefinition : STRING;
END_VAR
IF eStateMachine = RECIPES_MANAGER_IDLE THEN
	bReload := TRUE;
	bBusy := TRUE;
	bError := FALSE;
	iErrorId := 0;
	THIS^.sRecipesDefinition := sRecipesDefinition;
	THIS^.sRecipeName := sRecipeName;
	eStateMachine := RECIPES_MANAGER_RELOAD;
	MR_Reload := FALSE;
	fbMachineLogger.MR_AddLogs(CONCAT('Recipes_Manager',' : recipe reloading requested'));		
	
ELSIF eStateMachine = RECIPES_MANAGER_RELOAD_DONE THEN
	bReload := FALSE;
	bBusy := FALSE;
	MR_Reload := TRUE;
	fbMachineLogger.MR_AddLogs(CONCAT('Recipes_Manager',' : recipe reloading done'));
	
END_IF
END_METHOD

METHOD MR_ReloadExternal : BOOL
VAR_INPUT
	sRecipeName 			: STRING;
	sRecipesDefinition 		: STRING;
	sBackupStoragePath		: STRING;
END_VAR
IF eStateMachine = RECIPES_MANAGER_IDLE THEN
	bReload := TRUE;
	MR_ReloadExternal := FALSE;
	bBusy := TRUE;
	bError := FALSE;
	iErrorId := 0;
	THIS^.sRecipesDefinition := sRecipesDefinition;
	THIS^.sRecipeName := sRecipeName;
	THIS^.sBackupStoragePath := sBackupStoragePath;
	sStoragePath := sBackupStoragePath;
	M_SetStoragePath();
	eStateMachine := RECIPES_MANAGER_RELOAD;
	fbMachineLogger.MR_AddLogs(CONCAT('Recipes_Manager',' : recipe reloading requested'));		
	
ELSIF eStateMachine = RECIPES_MANAGER_RELOAD_DONE THEN
	sStoragePath := sLocalStoragePath;
	M_SetStoragePath();
	bReload := FALSE;
	bBusy := FALSE;
	MR_ReloadExternal := TRUE;
	fbMachineLogger.MR_AddLogs(CONCAT('Recipes_Manager',' : recipe reloading done'));
	
END_IF
END_METHOD

METHOD MR_Remove : BOOL
VAR_INPUT
	sRecipesDefinition : STRING;
	sRecipeName : STRING;
END_VAR
IF eStateMachine = RECIPES_MANAGER_IDLE THEN
	bRemove := TRUE;
	bBusy := TRUE;
	bError := FALSE;
	iErrorId := 0;
	THIS^.sRecipesDefinition := sRecipesDefinition;
	THIS^.sRecipeName := sRecipeName;
	M_ReloadRecipes();
	eStateMachine := RECIPES_MANAGER_REMOVE;
	eStateMachineCreateRemove := RECIPES_MANAGER_CREATE_REMOVE_OPERATION;
	fbMachineLogger.MR_AddLogs(CONCAT('Recipes_Manager',' : recipe removal requested'));	
	
ELSIF eStateMachine = RECIPES_MANAGER_REMOVE_DONE THEN
	bRemove := FALSE;
	bBusy := FALSE;
	MR_Remove := TRUE;
	fbMachineLogger.MR_AddLogs(CONCAT('Recipes_Manager',' : recipe removal done'));	
	
END_IF
END_METHOD

METHOD MR_Restore : BOOL
VAR_INPUT
	sRecipesDefinition		: STRING;
	sRecipeName				: STRING;
	sBackupStoragePath		: STRING;
END_VAR
IF eStateMachine = RECIPES_MANAGER_IDLE THEN
	bRestore := TRUE;
	bBusy := TRUE;
	bError := FALSE;
	iErrorId := 0;
	MR_Restore := FALSE;
	THIS^.sRecipesDefinition := sRecipesDefinition;
	THIS^.sRecipeName := sRecipeName;
	THIS^.sBackupStoragePath := sBackupStoragePath;
	sStoragePath := sBackupStoragePath;
	M_SetStoragePath();
	M_ReloadRecipes();
	eStateMachine := RECIPES_MANAGER_RESTORE;
	fbMachineLogger.MR_AddLogs(CONCAT('Recipes_Manager',' : recipe backup requested'));	
	
ELSIF eStateMachine = RECIPES_MANAGER_RESTORE_DONE THEN
	bRestore := FALSE;
	bBusy := FALSE;
	MR_Restore := TRUE;
	sStoragePath := sLocalStoragePath;
	M_SetStoragePath();
	fbMachineLogger.MR_AddLogs(CONCAT('Recipes_Manager',' : recipe backup done'));	
	
END_IF
END_METHOD

(*
When the command is executed, TwinCAT saves the values of the selected recipe in a file with the extension *.txtrecipe, whose name must be defined.
The standard dialog for saving a file opens. The format results from the settings of the Recipe Manager in the Storage tab.
*)
METHOD MR_Save : BOOL
VAR_INPUT
	sRecipesDefinition : STRING;
	sRecipeName : STRING;
END_VAR
IF eStateMachine = RECIPES_MANAGER_IDLE THEN
	bSave:= TRUE;
	bBusy := TRUE;
	bError := FALSE;
	iErrorId := 0;
	THIS^.sRecipesDefinition := sRecipesDefinition;
	THIS^.sRecipeName := sRecipeName;
	M_ReloadRecipes();
	eStateMachine := RECIPES_MANAGER_SAVE;
	fbMachineLogger.MR_AddLogs(CONCAT('Recipes_Manager',' : recipe save requested'));		
	
ELSIF eStateMachine = RECIPES_MANAGER_SAVE_DONE THEN
	bSave := FALSE;
	bBusy := FALSE;
	MR_Save := TRUE;
	fbMachineLogger.MR_AddLogs(CONCAT('Recipes_Manager',' : recipe save done'));	
	
END_IF
END_METHOD

METHOD MR_Writte : BOOL
VAR_INPUT
	sRecipesDefinition : STRING;
	sRecipeName : STRING;
END_VAR
IF eStateMachine = RECIPES_MANAGER_IDLE THEN
	bWrite := TRUE;
	bBusy := TRUE;
	bError := FALSE;
	iErrorId := 0;
	THIS^.sRecipesDefinition := sRecipesDefinition;
	THIS^.sRecipeName := sRecipeName;
	M_ReloadRecipes();
	eStateMachine := RECIPES_MANAGER_WRITE;
	fbMachineLogger.MR_AddLogs(CONCAT('Recipes_Manager',' : recipe writing requested'));		
	
ELSIF eStateMachine = RECIPES_MANAGER_WRITE_DONE THEN
	bWrite := FALSE;
	bBusy := FALSE;
	MR_Writte := TRUE;
	fbMachineLogger.MR_AddLogs(CONCAT('Recipes_Manager',' : recipe writing done'));	
	
END_IF
END_METHOD

METHOD PROTECTED MS_Aborting
VAR
	i: INT;
END_VAR
(* Reseting internal command bits*)
bInit				:= FALSE;
bCreate				:= FALSE;
bLoad				:= FALSE;
bLoadAndWrite		:= FALSE;
bRead				:= FALSE;
bReadAndSave		:= FALSE;
bRemove				:= FALSE;
bSave				:= FALSE;
bWrite				:= FALSE;
bGetRecipeCount		:= FALSE;
bGetNameArray		:= FALSE;
bGetVariableNames	:= FALSE;
bGetRecipeNames		:= FALSE;
bGetVariableValues	:= FALSE;
bReload				:= FALSE;
bRestore			:= FALSE;
bBackup				:= FALSE;

	
bActive	:= FALSE;
bBusy 	:= FALSE;
	
bLastSetStoragePathResult := FALSE;
iRecipesCount := 0;

FOR i := 0 TO iMAX_NUMBER_OF_RECIPES - 1 BY 1 DO
	MEMSET(ADR(arrVariableNames[i]),0,SIZEOF(arrVariableNames[i]));
END_FOR

FOR i := 0 TO iMAX_NUMBER_OF_VARIABLES_IN_RECIPES - 1 BY 1 DO
	MEMSET(ADR(arrRecipesNames[i]),0,SIZEOF(arrRecipesNames[i]));
END_FOR

FOR i := 0 TO iMAX_NUMBER_OF_VARIABLES_IN_RECIPES - 1 BY 1 DO
	MEMSET(ADR(arrRecipeValues[i]),0,SIZEOF(arrRecipeValues[i]));
END_FOR


eStateMachine := RECIPES_MANAGER_UNINITIALIZED;
END_METHOD

METHOD PROTECTED MS_Backup
CASE eStateMachineBackup OF
	RECIPES_MANAGER_BACKUP_OPERATION:	
		iLastResult := fbRecipeManager.CreateRecipe(sRecipesDefinition, sRecipeName);

		IF iLastResult = ERR_OK THEN
			eStateMachineBackup := RECIPES_MANAGER_BACKUP_RELOAD;
		ELSE
			bError := TRUE;
			iErrorId := fbRecipeManager.GetLastError();
			eStateMachine := RECIPES_MANAGER_BACKUP_DONE;
		END_IF
	
	RECIPES_MANAGER_BACKUP_RELOAD:
		iLastResult := fbRecipeManager.ReloadRecipes(sRecipesDefinition);
		
		IF iLastResult = ERR_OK THEN
			eStateMachineBackup := RECIPES_MANAGER_BACKUP_GET_RECIPES_COUNT;
		ELSE
			bError := TRUE;
			iErrorId := fbRecipeManager.GetLastError();
			eStateMachine := RECIPES_MANAGER_BACKUP_DONE;
		END_IF
		
	RECIPES_MANAGER_BACKUP_GET_RECIPES_COUNT:
		M_GetRecipesCount();
		
		IF iLastResult = ERR_OK THEN
			eStateMachineBackup := RECIPES_MANAGER_BACKUP_GET_RECIPES_NAMES;
		ELSE
			bError := TRUE;
			iErrorId := fbRecipeManager.GetLastError();
			eStateMachine := RECIPES_MANAGER_BACKUP_DONE;
		END_IF
	
	RECIPES_MANAGER_BACKUP_GET_RECIPES_NAMES:
		M_GetRecipesNames();
		
		IF iLastResult = ERR_OK THEN
			eStateMachineBackup := RECIPES_MANAGER_BACKUP_GET_VARIABLE_NAMES;
		ELSE
			bError := TRUE;
			iErrorId := fbRecipeManager.GetLastError();
			eStateMachine := RECIPES_MANAGER_BACKUP_DONE;
		END_IF
	
	RECIPES_MANAGER_BACKUP_GET_VARIABLE_NAMES:
		M_GetVariableNames();
		
		IF iLastResult = ERR_OK THEN
			eStateMachineBackup := RECIPES_MANAGER_BACKUP_GET_VARIABLE_VALUES;
		ELSE
			bError := TRUE;
			iErrorId := fbRecipeManager.GetLastError();
			eStateMachine := RECIPES_MANAGER_BACKUP_DONE;
		END_IF
		
	RECIPES_MANAGER_BACKUP_GET_VARIABLE_VALUES:
		M_GetVariableValues();
		
		IF iLastResult = ERR_OK THEN
			eStateMachineBackup := RECIPES_MANAGER_BACKUP_BACKUP_DONE;
		ELSE
			bError := TRUE;
			iErrorId := fbRecipeManager.GetLastError();
			eStateMachine := RECIPES_MANAGER_BACKUP_DONE;
		END_IF
	
	RECIPES_MANAGER_BACKUP_BACKUP_DONE:
		eStateMachineBackup := RECIPES_MANAGER_BACKUP_OPERATION;
		eStateMachine := RECIPES_MANAGER_BACKUP_DONE;
		
END_CASE
END_METHOD

METHOD PROTECTED MS_BackupDone
IF NOT bBackup THEN
	eStateMachine := RECIPES_MANAGER_IDLE;
	eStateMachineBackup := RECIPES_MANAGER_BACKUP_OPERATION;
END_IF
END_METHOD

METHOD PROTECTED MS_Create
CASE eStateMachineCreateRemove OF
	RECIPES_MANAGER_CREATE_REMOVE_OPERATION:	
		iLastResult := fbRecipeManager.CreateRecipe(sRecipesDefinition, sRecipeName);

		IF iLastResult = ERR_OK THEN
			eStateMachineCreateRemove := RECIPES_MANAGER_CREATE_REMOVE_RELOAD;
		ELSE
			bError := TRUE;
			iErrorId := fbRecipeManager.GetLastError();
			eStateMachine := RECIPES_MANAGER_CREATE_DONE;
		END_IF
	
	RECIPES_MANAGER_CREATE_REMOVE_RELOAD:
		iLastResult := fbRecipeManager.ReloadRecipes(sRecipesDefinition);
		
		IF iLastResult = ERR_OK THEN
			eStateMachineCreateRemove := RECIPES_MANAGER_CREATE_REMOVE_GET_RECIPES_COUNT;
		ELSE
			bError := TRUE;
			iErrorId := fbRecipeManager.GetLastError();
			eStateMachine := RECIPES_MANAGER_CREATE_DONE;
		END_IF
		
	RECIPES_MANAGER_CREATE_REMOVE_GET_RECIPES_COUNT:
		M_GetRecipesCount();
		
		IF iLastResult = ERR_OK THEN
			eStateMachineCreateRemove := RECIPES_MANAGER_CREATE_REMOVE_GET_RECIPES_NAMES;
		ELSE
			bError := TRUE;
			iErrorId := fbRecipeManager.GetLastError();
			eStateMachine := RECIPES_MANAGER_CREATE_DONE;
		END_IF
	
	RECIPES_MANAGER_CREATE_REMOVE_GET_RECIPES_NAMES:
		M_GetRecipesNames();
		
		IF iLastResult = ERR_OK THEN
			eStateMachineCreateRemove := RECIPES_MANAGER_CREATE_REMOVE_GET_VARIABLE_NAMES;
		ELSE
			bError := TRUE;
			iErrorId := fbRecipeManager.GetLastError();
			eStateMachine := RECIPES_MANAGER_CREATE_DONE;
		END_IF
	
	RECIPES_MANAGER_CREATE_REMOVE_GET_VARIABLE_NAMES:
		M_GetVariableNames();
		
		IF iLastResult = ERR_OK THEN
			eStateMachineCreateRemove := RECIPES_MANAGER_CREATE_REMOVE_GET_VARIABLE_VALUES;
		ELSE
			bError := TRUE;
			iErrorId := fbRecipeManager.GetLastError();
			eStateMachine := RECIPES_MANAGER_CREATE_DONE;
		END_IF
		
	RECIPES_MANAGER_CREATE_REMOVE_GET_VARIABLE_VALUES:
		M_GetVariableValues();
		
		IF iLastResult = ERR_OK THEN
			eStateMachineCreateRemove := RECIPES_MANAGER_CREATE_REMOVE_DONE;
		ELSE
			bError := TRUE;
			iErrorId := fbRecipeManager.GetLastError();
			eStateMachine := RECIPES_MANAGER_CREATE_DONE;
		END_IF
	
	RECIPES_MANAGER_CREATE_REMOVE_DONE:
		eStateMachineCreateRemove := RECIPES_MANAGER_CREATE_REMOVE_OPERATION;
		eStateMachine := RECIPES_MANAGER_CREATE_DONE;
		
END_CASE
END_METHOD

METHOD PROTECTED MS_CreateDone
IF NOT bCreate THEN
	eStateMachine := RECIPES_MANAGER_IDLE;
	eStateMachineCreateRemove := RECIPES_MANAGER_CREATE_REMOVE_OPERATION;
END_IF
END_METHOD

METHOD PROTECTED MS_GetRecipesNames
M_GetRecipesNames();
																								
IF iLastResult <> ERR_OK THEN
	bError := TRUE;
	iErrorId := fbRecipeManager.GetLastError();
END_IF
IF arrRecipesNames[iRecipesCount] <> '' THEN
	eStateMachine := RECIPES_MANAGER_GET_RECIPE_NAME_ARRAY_DONE;
END_IF
END_METHOD

METHOD PROTECTED MS_GetRecipesNamesDone
IF NOT bGetNameArray THEN
	eStateMachine := RECIPES_MANAGER_IDLE;
END_IF
END_METHOD

METHOD PROTECTED MS_GetVariableNames
M_GetVariableNames();
																								
IF iLastResult <> ERR_OK THEN
	bError := TRUE;
	iErrorId := fbRecipeManager.GetLastError();
END_IF

eStateMachine := RECIPES_MANAGER_GET_RECIPE_VARIABLE_NAMES_DONE;
END_METHOD

METHOD PROTECTED MS_GetVariableNamesDone
IF NOT bGetVariableNames THEN
	eStateMachine := RECIPES_MANAGER_IDLE;
END_IF
END_METHOD

METHOD PROTECTED MS_GetVariableValues
VAR_INPUT
END_VAR
M_GetVariableValues();

IF iLastResult <> ERR_OK THEN
	bError := TRUE;
	iErrorId := fbRecipeManager.GetLastError();
END_IF

eStateMachine := RECIPES_MANAGER_GET_RECIPE_VARIABLE_VALUES_DONE;
END_METHOD

METHOD PROTECTED MS_GetVariableValuesDone
IF NOT bGetVariableValues THEN
	eStateMachine := RECIPES_MANAGER_READ;
END_IF
END_METHOD

METHOD PROTECTED MS_Idle
;
END_METHOD

METHOD PROTECTED MS_Initialization
CASE eStateMachineInit OF
    RECIPES_MANAGER_INIT_SET_STORAGE_PATH:
		sStoragePath := sLocalStoragePath;
        M_SetStoragePath(); 
        
        IF bLastSetStoragePathResult THEN
            eStateMachineInit := RECIPES_MANAGER_INIT_RELOAD;
        ELSE
            bError  := TRUE;
            iErrorId := fbRecipeManager.GetLastError();
            eStateMachine := RECIPES_MANAGER_ABORTING;
        END_IF
        
    RECIPES_MANAGER_INIT_RELOAD:
        M_ReloadRecipes();
        
        IF iLastResult = ERR_OK THEN
            eStateMachineInit := RECIPES_MANAGER_INIT_GET_RECIPES_COUNT;
        ELSE
            bError  := TRUE;
            iErrorId := fbRecipeManager.GetLastError();
            eStateMachine := RECIPES_MANAGER_ABORTING;
        END_IF
    
    RECIPES_MANAGER_INIT_GET_RECIPES_COUNT:
        M_GetRecipesCount();
        
        IF iLastResult = ERR_OK THEN
            eStateMachineInit := RECIPES_MANAGER_INIT_GET_RECIPES_NAMES;
        ELSE
            bError  := TRUE;
            iErrorId := fbRecipeManager.GetLastError();
            eStateMachine := RECIPES_MANAGER_ABORTING;
        END_IF
    
    RECIPES_MANAGER_INIT_GET_RECIPES_NAMES:
        M_GetRecipesNames();
                                                            
        IF iLastResult = ERR_OK THEN
            eStateMachineInit := RECIPES_MANAGER_INIT_DONE;
        ELSE
            bError  := TRUE;
            iErrorId := fbRecipeManager.GetLastError();
            eStateMachine := RECIPES_MANAGER_ABORTING;
        END_IF
    (*
	(* Not included because removing all recipes from device memory will result error occurring *)
    RECIPES_MANAGER_INIT_GET_VARIABLE_NAMES:
	    M_GetVariableNames(); 
                                                                
        IF iLastResult = ERR_OK THEN
            eStateMachineInit := RECIPES_MANAGER_INIT_GET_VARIABLE_VALUES;
        ELSE
            bError  := TRUE;
           iErrorId := fbRecipeManager.GetLastError();
            eStateMachine := RECIPES_MANAGER_ABORTING;
        END_IF
    
    RECIPES_MANAGER_INIT_GET_VARIABLE_VALUES:
        M_GetVariableValues(); //
                                                        
        IF iLastResult = ERR_OK THEN
            eStateMachineInit := RECIPES_MANAGER_INIT_DONE;
        ELSE
            bError  := TRUE;
            iErrorId := fbRecipeManager.GetLastError();
            eStateMachine := RECIPES_MANAGER_ABORTING;
        END_IF
    *)
	
    RECIPES_MANAGER_INIT_DONE:
		eStateMachineInit := RECIPES_MANAGER_INIT_SET_STORAGE_PATH;
        eStateMachine := RECIPES_MANAGER_IDLE;
    
END_CASE
END_METHOD

METHOD PROTECTED MS_Load
iLastResult := fbRecipeManager.LoadRecipe(sRecipesDefinition, sRecipeName);

IF iLastResult <> ERR_OK THEN
	bError := TRUE;
	iErrorId := fbRecipeManager.GetLastError();
END_IF

eStateMachine := RECIPES_MANAGER_LOAD_DONE;
END_METHOD

METHOD PROTECTED MS_LoadDone
IF NOT bLoad THEN
	eStateMachine := RECIPES_MANAGER_IDLE;
END_IF
END_METHOD

METHOD PROTECTED MS_LoadWritte
iLastResult := fbRecipeManager.LoadAndWriteRecipe(sRecipesDefinition, sRecipeName);

IF iLastResult <> ERR_OK THEN
	bError := TRUE;
	iErrorId := fbRecipeManager.GetLastError();
END_IF

eStateMachine := RECIPES_MANAGER_LOAD_AND_WRITE_DONE;
END_METHOD

METHOD PROTECTED MS_LoadWritteDone
IF NOT bLoadAndWrite THEN
	eStateMachine := RECIPES_MANAGER_IDLE;
END_IF
END_METHOD

METHOD PROTECTED MS_Read
iLastResult := fbRecipeManager.ReadRecipe(sRecipesDefinition, sRecipeName);

IF iLastResult <> ERR_OK THEN
	bError := TRUE;
	iErrorId := fbRecipeManager.GetLastError();
END_IF

eStateMachine := RECIPES_MANAGER_READ_DONE;
END_METHOD

METHOD PROTECTED MS_ReadDone
IF NOT bRead THEN
	eStateMachine := RECIPES_MANAGER_IDLE;
END_IF
END_METHOD

METHOD PROTECTED MS_ReadSave
iLastResult := fbRecipeManager.ReadAndSaveRecipe(sRecipesDefinition, sRecipeName);

IF iLastResult <> ERR_OK THEN
	bError := TRUE;
	iErrorId := fbRecipeManager.GetLastError();
END_IF

eStateMachine := RECIPES_MANAGER_READ_AND_SAVE_DONE;
END_METHOD

METHOD PROTECTED MS_ReadSaveDone
IF NOT bReadAndSave THEN
	eStateMachine := RECIPES_MANAGER_IDLE;
END_IF
END_METHOD

METHOD PROTECTED MS_Reload
VAR_INPUT
END_VAR
CASE eStateMachineReload OF
	RECIPE_MANAGER_RELOAD_OPERATION:
		iLastResult := fbRecipeManager.ReloadRecipes(sRecipesDefinition);
		
		IF iLastResult = ERR_OK THEN
			eStateMachineReload := RECIPE_MANAGER_RELOAD_GET_RECIPES_COUNT;
		ELSE
			bError := TRUE;
			iErrorId := fbRecipeManager.GetLastError();
			eStateMachine := RECIPES_MANAGER_RELOAD_DONE;
		END_IF
		
	RECIPE_MANAGER_RELOAD_GET_RECIPES_COUNT:
		M_GetRecipesCount();
		
		IF iLastResult = ERR_OK THEN
			eStateMachineReload := RECIPE_MANAGER_RELOAD_GET_RECIPES_NAMES;
		ELSE
			bError := TRUE;
			iErrorId := fbRecipeManager.GetLastError();
			eStateMachine := RECIPES_MANAGER_RELOAD_DONE;
		END_IF
	
	RECIPE_MANAGER_RELOAD_GET_RECIPES_NAMES:
		M_GetRecipesNames();
		
		IF iLastResult = ERR_OK THEN
			eStateMachineReload := RECIPE_MANAGER_RELOAD_GET_VARIABLE_NAMES;
		ELSE
			bError := TRUE;
			iErrorId := fbRecipeManager.GetLastError();
			eStateMachine := RECIPES_MANAGER_RELOAD_DONE;
		END_IF
	
	RECIPE_MANAGER_RELOAD_GET_VARIABLE_NAMES:
		M_GetVariableNames();
		
		IF iLastResult = ERR_OK THEN
			eStateMachineReload := RECIPE_MANAGER_RELOAD_GET_VARIABLE_VALUES;
		ELSE
			bError := TRUE;
			iErrorId := fbRecipeManager.GetLastError();
			eStateMachine := RECIPES_MANAGER_RELOAD_DONE;
		END_IF
		
	RECIPE_MANAGER_RELOAD_GET_VARIABLE_VALUES:
		M_GetVariableValues();
		
		IF iLastResult = ERR_OK THEN
			eStateMachineReload := RECIPE_MANAGER_RELOAD_DONE;
		ELSE
			bError := TRUE;
			iErrorId := fbRecipeManager.GetLastError();
			eStateMachine := RECIPES_MANAGER_RELOAD_DONE;
		END_IF
	
	RECIPE_MANAGER_RELOAD_DONE:
		eStateMachineReload := RECIPE_MANAGER_RELOAD_OPERATION;
		eStateMachine := RECIPES_MANAGER_RELOAD_DONE;
		
END_CASE
END_METHOD

METHOD PROTECTED MS_ReloadDone
VAR_INPUT
END_VAR
IF NOT bReload THEN
	eStateMachine := RECIPES_MANAGER_IDLE;
END_IF
END_METHOD

METHOD PROTECTED MS_Remove
CASE eStateMachineCreateRemove OF
	RECIPES_MANAGER_CREATE_REMOVE_OPERATION:
		iLastResult := fbRecipeManager.DeleteRecipe(sRecipesDefinition, sRecipeName);

		IF iLastResult = ERR_OK THEN
			eStateMachineCreateRemove := RECIPES_MANAGER_CREATE_REMOVE_RELOAD;
		ELSE
			bError := TRUE;
			iErrorId := fbRecipeManager.GetLastError();
			eStateMachine := RECIPES_MANAGER_REMOVE_DONE;
		END_IF
	
	RECIPES_MANAGER_CREATE_REMOVE_RELOAD:
		iLastResult := fbRecipeManager.ReloadRecipes(sRecipesDefinition);
		
		IF iLastResult = ERR_OK THEN
			eStateMachineCreateRemove := RECIPES_MANAGER_CREATE_REMOVE_GET_RECIPES_COUNT;
		ELSE
			bError := TRUE;
			iErrorId := fbRecipeManager.GetLastError();
			eStateMachine := RECIPES_MANAGER_REMOVE_DONE;
		END_IF
		
	RECIPES_MANAGER_CREATE_REMOVE_GET_RECIPES_COUNT:
		M_GetRecipesCount();
		
		IF iLastResult = ERR_OK THEN
			eStateMachineCreateRemove := RECIPES_MANAGER_CREATE_REMOVE_GET_RECIPES_NAMES;
		ELSE
			bError := TRUE;
			iErrorId := fbRecipeManager.GetLastError();
			eStateMachine := RECIPES_MANAGER_REMOVE_DONE;
		END_IF
	
	RECIPES_MANAGER_CREATE_REMOVE_GET_RECIPES_NAMES:
		M_GetRecipesNames();
		
		IF iLastResult = ERR_OK THEN
			eStateMachineCreateRemove := RECIPES_MANAGER_CREATE_REMOVE_GET_VARIABLE_NAMES;
		ELSE
			bError := TRUE;
			iErrorId := fbRecipeManager.GetLastError();
			eStateMachine := RECIPES_MANAGER_REMOVE_DONE;
		END_IF
	
	RECIPES_MANAGER_CREATE_REMOVE_GET_VARIABLE_NAMES:
		M_GetVariableNames();
		
		IF iLastResult = ERR_OK THEN
			eStateMachineCreateRemove := RECIPES_MANAGER_CREATE_REMOVE_GET_VARIABLE_VALUES;
		ELSE
			bError := TRUE;
			iErrorId := fbRecipeManager.GetLastError();
			eStateMachine := RECIPES_MANAGER_REMOVE_DONE;
		END_IF
		
	RECIPES_MANAGER_CREATE_REMOVE_GET_VARIABLE_VALUES:
		M_GetVariableValues();
		
		IF iLastResult = ERR_OK THEN
			eStateMachineCreateRemove := RECIPES_MANAGER_CREATE_REMOVE_DONE;
		ELSE
			bError := TRUE;
			iErrorId := fbRecipeManager.GetLastError();
			eStateMachine := RECIPES_MANAGER_REMOVE_DONE;
		END_IF
	
	RECIPES_MANAGER_CREATE_REMOVE_DONE:
		eStateMachineCreateRemove := RECIPES_MANAGER_CREATE_REMOVE_OPERATION;
		eStateMachine := RECIPES_MANAGER_REMOVE_DONE;
		
END_CASE
END_METHOD

METHOD PROTECTED MS_RemoveDone
IF NOT bRemove THEN
	eStateMachineCreateRemove := RECIPES_MANAGER_CREATE_REMOVE_OPERATION;
	eStateMachine := RECIPES_MANAGER_IDLE;
END_IF
END_METHOD

METHOD PROTECTED MS_Restore
iLastResult := fbRecipeManager.LoadAndWriteRecipe(sRecipesDefinition, sRecipeName);

IF iLastResult <> ERR_OK THEN
	bError := TRUE;
	iErrorId := fbRecipeManager.GetLastError();
END_IF

eStateMachine := RECIPES_MANAGER_RESTORE_DONE;
END_METHOD

METHOD PROTECTED MS_RestoreDone
IF NOT bRestore THEN
	eStateMachine := RECIPES_MANAGER_IDLE;
END_IF
END_METHOD

METHOD PROTECTED MS_Save
iLastResult := fbRecipeManager.SaveRecipe(sRecipesDefinition, sRecipeName);

IF iLastResult <> ERR_OK THEN
	bError := TRUE;
	iErrorId := fbRecipeManager.GetLastError();
END_IF

eStateMachine := RECIPES_MANAGER_SAVE_DONE;
END_METHOD

METHOD PROTECTED MS_SaveDone
IF NOT bSave THEN
	eStateMachine := RECIPES_MANAGER_IDLE;
END_IF
END_METHOD

METHOD PROTECTED MS_Uninitialized
VAR
	i: INT;
END_VAR
END_METHOD

METHOD PROTECTED MS_Writte
iLastResult := fbRecipeManager.WriteRecipe(sRecipesDefinition, sRecipeName);

IF iLastResult <> ERR_OK THEN
	bError := TRUE;
	iErrorId := fbRecipeManager.GetLastError();
END_IF

eStateMachine := RECIPES_MANAGER_WRITE_DONE;
END_METHOD

METHOD PROTECTED MS_WritteDone
IF NOT bWrite THEN
	eStateMachine := RECIPES_MANAGER_IDLE;
END_IF
END_METHOD

PROPERTY RecipeCount : REFERENCE TO USINT
GET
RecipeCount REF= iRecipesCount;
END_GET
END_PROPERTY

PROPERTY RecipesDefinition : REFERENCE TO STRING
GET
RecipesDefinition REF= sRecipesDefinition;
END_GET
END_PROPERTY

PROPERTY RecipesNames : REFERENCE TO ARRAY	[0..iMAX_NUMBER_OF_RECIPES-1] OF STRING;
GET
RecipesNames REF= arrRecipesNames;
END_GET
END_PROPERTY

PROPERTY RecipeValues : REFERENCE TO ARRAY [0..iMAX_NUMBER_OF_VARIABLES_IN_RECIPES-1] OF STRING
//PROPERTY RecipeValues : ARRAY [0..iMAX_NUMBER_OF_VARIABLES_IN_RECIPES-1] OF STRING(iMAX_RECIPE_NAME_LENGTH)
GET
RecipeValues REF= arrRecipeValues;
END_GET
END_PROPERTY

PROPERTY RecipeValuesAdr : REFERENCE TO ARRAY [0..iMAX_NUMBER_OF_VARIABLES_IN_RECIPES-1] OF PVOID
GET
RecipeValuesAdr REF= arrRecipeValuesAdr;
END_GET
END_PROPERTY

PROPERTY RecipeValuesAdrAvailable : REFERENCE TO BOOL
GET
RecipeValuesAdrAvailable REF= bRecipeFileValuesAdrAvailable;
END_GET
END_PROPERTY

PROPERTY State : REFERENCE TO E_RecipesManagerState;
GET
State REF= eStateMachine;
END_GET
END_PROPERTY

METHOD PROTECTED StateMachine
CASE eStateMachine OF
	RECIPES_MANAGER_UNINITIALIZED:
		MS_Uninitialized();
		
	RECIPES_MANAGER_INITIALIZATION:
		MS_Initialization();
		
	RECIPES_MANAGER_IDLE:
		MS_Idle();
		
	RECIPES_MANAGER_CREATE:
		MS_Create();
		
	RECIPES_MANAGER_CREATE_DONE:
		MS_CreateDone();
		
	RECIPES_MANAGER_REMOVE:
		MS_Remove();
		
	RECIPES_MANAGER_REMOVE_DONE:
		MS_RemoveDone();
		
	RECIPES_MANAGER_LOAD:
		MS_Load();
		
	RECIPES_MANAGER_LOAD_DONE:
		MS_LoadDone();
		
	RECIPES_MANAGER_SAVE:
		MS_Save();
		
	RECIPES_MANAGER_SAVE_DONE:
		MS_SaveDone();
		
	RECIPES_MANAGER_READ:
		MS_Read();
		
	RECIPES_MANAGER_READ_DONE:
		MS_ReadDone();	
	
	RECIPES_MANAGER_READ_AND_SAVE:
		MS_ReadSave();
	
	RECIPES_MANAGER_READ_AND_SAVE_DONE:
		MS_ReadSaveDone();
	
	RECIPES_MANAGER_WRITE:
		MS_Writte();
	
	RECIPES_MANAGER_WRITE_DONE:
		MS_WritteDone();
	
	RECIPES_MANAGER_LOAD_AND_WRITE:
		MS_LoadWritte();
	
	RECIPES_MANAGER_LOAD_AND_WRITE_DONE:
		MS_LoadWritteDone();
		
	RECIPES_MANAGER_GET_RECIPE_NAME_ARRAY:
		MS_GetRecipesNames();
	
	RECIPES_MANAGER_GET_RECIPE_NAME_ARRAY_DONE:
		MS_GetRecipesNamesDone();
		
	RECIPES_MANAGER_GET_RECIPE_VARIABLE_NAMES:
		MS_GetVariableNames();
	
	RECIPES_MANAGER_GET_RECIPE_VARIABLE_NAMES_DONE:
		MS_GetVariableNamesDone();
		
	RECIPES_MANAGER_GET_RECIPE_VARIABLE_VALUES:
		MS_GetVariableValues();
	
	RECIPES_MANAGER_GET_RECIPE_VARIABLE_VALUES_DONE:
		MS_GetVariableValuesDone();
		
	RECIPES_MANAGER_RELOAD:
		MS_Reload();
	
	RECIPES_MANAGER_RELOAD_DONE:
		MS_ReloadDone();
	
	RECIPES_MANAGER_BACKUP:
		MS_Backup();
	
	RECIPES_MANAGER_BACKUP_DONE:
		MS_BackupDone();
		
	RECIPES_MANAGER_RESTORE:
		MS_Restore();
	
	RECIPES_MANAGER_RESTORE_DONE:
		MS_RestoreDone();
		
	RECIPES_MANAGER_ABORTING:
		MS_Aborting();
	
END_CASE
END_METHOD

END_FUNCTION_BLOCK

// ---- POUs/Machine/Visu Control/PRG_VisuControl.TcPOU
PROGRAM PRG_VisuControl
VAR
	iLoop 			: USINT;			(*  *)
	bFirstCycle 	: BOOL := TRUE;		(*  *)
	fbVisuControl	: FB_VisuControl;	(*  *)
END_VAR

IF bFirstCycle AND stShell.stFlags.bMachineCtrlAssignamentsDone AND stShell.stFlags.bAlarmCtrlAssignamentsDone AND stShell.stFlags.bRecipesCtrlAssignamentsDone THEN
	bFirstCycle := FALSE;
	
	fbVisuControl.MR_FirstCycle( 	sMachineName 		:= sMACHINE_NAME,
									sSoftwareVersion	:= sSOFTWARE_VERSION);
									
	(*--- Append platform objects to HMI ---*)
	(* Apped machine controler to HMI controler *)
	fbVisuControl.MR_AppendUniversalMachine(ifMachine := stShell.stPlatform.ref_fbMachineControler);
	
	(* Append alarm controler to HMI controler *)
	fbVisuControl.MR_AppendAlarmControler(ifAlarmControler := stShell.stPlatform.ref_fbAlarmControler);
	
	(* Append recipes manager to HMI controler *)
	fbVisuControl.MR_AppendRecipesManager(ifRecipesManager := stShell.stPlatform.ref_fbRecipesManager);
	
	(* --- Append recipes parameters --- *)
	fbVisuControl.MR_AppendRecipeParameter( ifRecipeParameter := stShell.stRecipeData.rpVar1);
	fbVisuControl.MR_AppendRecipeParameter( ifRecipeParameter := stShell.stRecipeData.rpVar2);
	fbVisuControl.MR_AppendRecipeParameter( ifRecipeParameter := stShell.stRecipeData.rpVar3);
	fbVisuControl.MR_AppendRecipeParameter( ifRecipeParameter := stShell.stRecipeData.rpVar4);
	fbVisuControl.MR_AppendRecipeParameter( ifRecipeParameter := stShell.stRecipeData.rpVar5);
	fbVisuControl.MR_AppendRecipeParameter( ifRecipeParameter := stShell.stRecipeData.rpVar6);
	fbVisuControl.MR_AppendRecipeParameter( ifRecipeParameter := stShell.stRecipeData.rpVar7);
	fbVisuControl.MR_AppendRecipeParameter( ifRecipeParameter := stShell.stRecipeData.rpVar8);
	fbVisuControl.MR_AppendRecipeParameter( ifRecipeParameter := stShell.stRecipeData.rpVar9);
	fbVisuControl.MR_AppendRecipeParameter( ifRecipeParameter := stShell.stRecipeData.rpVar10);
	
	(* --- Append machine objects to HMI ---*)
//	(* Append sample digital inputs *)
//	FOR iLoop := 0 TO 19 DO
//		fbVisuControl.MR_AppendInput(ifDigitalInput := stShell.stPlatform.ref_fbMachineControler.Inputs[iLoop]);
//	END_FOR
	
//	(* Append sample digital outputs *)
//	FOR iLoop := 0 TO 19 DO
//		fbVisuControl.MR_AppendOutput(ifDigitalOutput := stShell.stPlatform.ref_fbMachineControler.Outputs[iLoop]);
//	END_FOR
	
